LIN {X 0,Y 525.406,Z 288.21,A -85,B 0,C 180,E1 -4793.658,E2 -4793.658} C_VEL
LIN {X 0,Y 523.939,Z 280.222,A -85,B 0,C 180,E1 -4794.968,E2 -4794.968} C_VEL
LIN {X 0,Y 523.912,Z 280.228,A -85,B 0,C 180,E1 -4798.002,E2 -4798.002} C_VEL
LIN {X 0,Y 523.934,Z 280.223,A -85,B 0,C 180,E1 -4800.852,E2 -4800.852} C_VEL
LIN {X 0,Y 523.928,Z 280.222,A -85,B 0,C 180,E1 -4803.729,E2 -4803.729} C_VEL
LIN {X 0,Y 523.897,Z 280.231,A -85,B 0,C 180,E1 -4806.4,E2 -4806.4} C_VEL
LIN {X 0,Y 523.911,Z 280.22,A -85,B 0,C 180,E1 -4809.085,E2 -4809.085} C_VEL
LIN {X 0,Y 523.949,Z 280.218,A -85,B 0,C 180,E1 -4812.119,E2 -4812.119} C_VEL
LIN {X 0,Y 523.941,Z 280.216,A -85,B 0,C 180,E1 -4815.31,E2 -4815.31} C_VEL
LIN {X 0,Y 523.953,Z 280.22,A -85,B 0,C 180,E1 -4818.689,E2 -4818.689} C_VEL
LIN {X 0,Y 523.915,Z 280.22,A -85,B 0,C 180,E1 -4821.08,E2 -4821.08} C_VEL
LIN {X 0,Y 523.897,Z 280.221,A -85,B 0,C 180,E1 -4823.825,E2 -4823.825} C_VEL
LIN {X 0,Y 523.91,Z 280.227,A -85,B 0,C 180,E1 -4826.633,E2 -4826.633} C_VEL
LIN {X 0,Y 523.953,Z 280.214,A -85,B 0,C 180,E1 -4829.355,E2 -4829.355} C_VEL
LIN {X 0,Y 523.975,Z 280.213,A -85,B 0,C 180,E1 -4832.281,E2 -4832.281} C_VEL
LIN {X 0,Y 523.944,Z 280.223,A -85,B 0,C 180,E1 -4834.581,E2 -4834.581} C_VEL
LIN {X 0,Y 523.916,Z 280.218,A -85,B 0,C 180,E1 -4837.756,E2 -4837.756} C_VEL
LIN {X 0,Y 523.973,Z 280.213,A -85,B 0,C 180,E1 -4840.408,E2 -4840.408} C_VEL
LIN {X 0,Y 523.965,Z 280.219,A -85,B 0,C 180,E1 -4842.837,E2 -4842.837} C_VEL
LIN {X 0,Y 523.974,Z 280.214,A -85,B 0,C 180,E1 -4845.236,E2 -4845.236} C_VEL
LIN {X 0,Y 524.009,Z 280.208,A -85,B 0,C 180,E1 -4848.394,E2 -4848.394} C_VEL
LIN {X 0,Y 524.001,Z 280.207,A -85,B 0,C 180,E1 -4851.516,E2 -4851.516} C_VEL
LIN {X 0,Y 524.078,Z 280.204,A -85,B 0,C 180,E1 -4854.614,E2 -4854.614} C_VEL
LIN {X 0,Y 524.11,Z 280.194,A -85,B 0,C 180,E1 -4857.695,E2 -4857.695} C_VEL
LIN {X 0,Y 524.121,Z 280.199,A -85,B 0,C 180,E1 -4860.769,E2 -4860.769} C_VEL
LIN {X 0,Y 524.069,Z 280.206,A -85,B 0,C 180,E1 -4863.075,E2 -4863.075} C_VEL
LIN {X 0,Y 524.043,Z 280.202,A -85,B 0,C 180,E1 -4866.159,E2 -4866.159} C_VEL
LIN {X 0,Y 523.996,Z 280.213,A -85,B 0,C 180,E1 -4869.262,E2 -4869.262} C_VEL
LIN {X 0,Y 524,Z 280.208,A -85,B 0,C 180,E1 -4871.74,E2 -4871.74} C_VEL
LIN {X 0,Y 523.991,Z 280.217,A -85,B 0,C 180,E1 -4875.053,E2 -4875.053} C_VEL
LIN {X 0,Y 523.945,Z 280.214,A -85,B 0,C 180,E1 -4877.97,E2 -4877.97} C_VEL
LIN {X 0,Y 523.97,Z 280.212,A -85,B 0,C 180,E1 -4880.41,E2 -4880.41} C_VEL
LIN {X 0,Y 523.908,Z 280.224,A -85,B 0,C 180,E1 -4882.894,E2 -4882.894} C_VEL
LIN {X 0,Y 523.981,Z 280.21,A -85,B 0,C 180,E1 -4886.02,E2 -4886.02} C_VEL
LIN {X 0,Y 523.927,Z 280.221,A -85,B 0,C 180,E1 -4888.876,E2 -4888.876} C_VEL
LIN {X 0,Y 523.917,Z 280.221,A -85,B 0,C 180,E1 -4891.545,E2 -4891.545} C_VEL
LIN {X 0,Y 523.921,Z 280.217,A -85,B 0,C 180,E1 -4894.292,E2 -4894.292} C_VEL
LIN {X 0,Y 523.906,Z 280.226,A -85,B 0,C 180,E1 -4897.133,E2 -4897.133} C_VEL
LIN {X 0,Y 523.937,Z 280.216,A -85,B 0,C 180,E1 -4900.13,E2 -4900.13} C_VEL
LIN {X 0,Y 523.889,Z 280.229,A -85,B 0,C 180,E1 -4903.171,E2 -4903.171} C_VEL
LIN {X 0,Y 523.923,Z 280.222,A -85,B 0,C 180,E1 -4905.771,E2 -4905.771} C_VEL
LIN {X 0,Y 523.885,Z 280.225,A -85,B 0,C 180,E1 -4906.911,E2 -4906.911} C_VEL
LIN {X 0,Y 523.209,Z 280.314,A -85,B 0,C 180,E1 -4907.553,E2 -4907.553} C_VEL
LIN {X 0,Y 520.362,Z 280.666,A -85,B 0,C 180,E1 -4908.594,E2 -4908.594} C_VEL
LIN {X 0,Y 517.964,Z 280.968,A -85,B 0,C 180,E1 -4909.433,E2 -4909.433} C_VEL
LIN {X 0,Y 516.939,Z 281.09,A -85,B 0,C 180,E1 -4910.081,E2 -4910.081} C_VEL
LIN {X 0,Y 516.858,Z 281.099,A -85,B 0,C 180,E1 -4910.3,E2 -4910.3} C_VEL
LIN {X 0,Y 516.846,Z 281.107,A -85,B 0,C 180,E1 -4913.349,E2 -4913.349} C_VEL
LIN {X 0,Y 516.884,Z 281.097,A -85,B 0,C 180,E1 -4916.12,E2 -4916.12} C_VEL
LIN {X 0,Y 516.882,Z 281.099,A -85,B 0,C 180,E1 -4918.939,E2 -4918.939} C_VEL
LIN {X 0,Y 516.958,Z 281.096,A -85,B 0,C 180,E1 -4922.172,E2 -4922.172} C_VEL
LIN {X 0,Y 517.261,Z 286.094,A -85,B 0,C 180,E1 -4923.144,E2 -4923.144} C_VEL
LIN {X 0,Y 517.143,Z 299.715,A -85,B 0,C 180,E1 -4925.679,E2 -4925.679} C_VEL
LIN {X 0,Y 519.184,Z 310.941,A -85,B 0,C 180,E1 -4925.909,E2 -4925.909} C_VEL
LIN {X 0,Y 518.63,Z 406.558,A -85,B 0,C 180,E1 -4927.253,E2 -4927.253} C_VEL
LIN {X 0,Y 518.525,Z 420.061,A -85,B 0,C 180,E1 -4927.608,E2 -4927.608} C_VEL
LIN {X 0,Y 518.216,Z 432.786,A -85,B 0,C 180,E1 -4928.103,E2 -4928.103} C_VEL
LIN {X 0,Y 517.976,Z 444.369,A -85,B 0,C 180,E1 -4928.719,E2 -4928.719} C_VEL
LIN {X 0,Y 517.646,Z 456.07,A -85,B 0,C 180,E1 -4929.523,E2 -4929.523} C_VEL
LIN {X 0,Y 517.317,Z 466.867,A -85,B 0,C 180,E1 -4930.456,E2 -4930.456} C_VEL
LIN {X 0,Y 517.068,Z 475.452,A -85,B 0,C 180,E1 -4931.373,E2 -4931.373} C_VEL
LIN {X 0,Y 516.808,Z 484.688,A -85,B 0,C 180,E1 -4932.592,E2 -4932.592} C_VEL
LIN {X 0,Y 516.604,Z 492.063,A -85,B 0,C 180,E1 -4933.807,E2 -4933.807} C_VEL
LIN {X 0,Y 516.469,Z 498.021,A -85,B 0,C 180,E1 -4935.052,E2 -4935.052} C_VEL
LIN {X 0,Y 516.366,Z 502.404,A -85,B 0,C 180,E1 -4936.221,E2 -4936.221} C_VEL
LIN {X 0,Y 516.297,Z 505.806,A -85,B 0,C 180,E1 -4937.421,E2 -4937.421} C_VEL
LIN {X 0,Y 516.285,Z 508.091,A -85,B 0,C 180,E1 -4938.556,E2 -4938.556} C_VEL
LIN {X 0,Y 516.239,Z 509.597,A -85,B 0,C 180,E1 -4939.807,E2 -4939.807} C_VEL
LIN {X 0,Y 516.233,Z 510.026,A -85,B 0,C 180,E1 -4941.388,E2 -4941.388} C_VEL
LIN {X 0,Y 516.273,Z 509.658,A -85,B 0,C 180,E1 -4942.177,E2 -4942.177} C_VEL
LIN {X 0,Y 516.32,Z 508.057,A -85,B 0,C 180,E1 -4943.547,E2 -4943.547} C_VEL
LIN {X 0,Y 516.32,Z 506.098,A -85,B 0,C 180,E1 -4944.533,E2 -4944.533} C_VEL
LIN {X 0,Y 516.361,Z 502.896,A -85,B 0,C 180,E1 -4945.707,E2 -4945.707} C_VEL
LIN {X 0,Y 516.434,Z 498.648,A -85,B 0,C 180,E1 -4946.88,E2 -4946.88} C_VEL
LIN {X 0,Y 516.584,Z 492.239,A -85,B 0,C 180,E1 -4948.246,E2 -4948.246} C_VEL
LIN {X 0,Y 516.817,Z 485.213,A -85,B 0,C 180,E1 -4949.416,E2 -4949.416} C_VEL
LIN {X 0,Y 517.049,Z 476.502,A -85,B 0,C 180,E1 -4950.585,E2 -4950.585} C_VEL
LIN {X 0,Y 517.306,Z 466.62,A -85,B 0,C 180,E1 -4951.655,E2 -4951.655} C_VEL
LIN {X 0,Y 517.543,Z 456.543,A -85,B 0,C 180,E1 -4952.53,E2 -4952.53} C_VEL
LIN {X 0,Y 517.832,Z 445.389,A -85,B 0,C 180,E1 -4953.307,E2 -4953.307} C_VEL
LIN {X 0,Y 518.125,Z 434.797,A -85,B 0,C 180,E1 -4953.889,E2 -4953.889} C_VEL
LIN {X 0,Y 518.308,Z 423.339,A -85,B 0,C 180,E1 -4954.375,E2 -4954.375} C_VEL
LIN {X 0,Y 518.512,Z 411.153,A -85,B 0,C 180,E1 -4954.738,E2 -4954.738} C_VEL
LIN {X 0,Y 518.632,Z 395.767,A -85,B 0,C 180,E1 -4955.005,E2 -4955.005} C_VEL
LIN {X 0,Y 519.17,Z 310.059,A -85,B 0,C 180,E1 -4956.193,E2 -4956.193} C_VEL
LIN {X 0,Y 517.205,Z 299.754,A -85,B 0,C 180,E1 -4956.416,E2 -4956.416} C_VEL
LIN {X 0,Y 517.361,Z 285.225,A -85,B 0,C 180,E1 -4959.185,E2 -4959.185} C_VEL
LIN {X 0,Y 516.873,Z 281.104,A -85,B 0,C 180,E1 -4960.033,E2 -4960.033} C_VEL
LIN {X 0,Y 516.906,Z 281.1,A -85,B 0,C 180,E1 -4962.565,E2 -4962.565} C_VEL
LIN {X 0,Y 516.892,Z 281.093,A -85,B 0,C 180,E1 -4965.78,E2 -4965.78} C_VEL
LIN {X 0,Y 516.878,Z 281.097,A -85,B 0,C 180,E1 -4968.224,E2 -4968.224} C_VEL
LIN {X 0,Y 516.907,Z 281.1,A -85,B 0,C 180,E1 -4970.702,E2 -4970.702} C_VEL
LIN {X 0,Y 516.862,Z 281.1,A -85,B 0,C 180,E1 -4973.224,E2 -4973.224} C_VEL
LIN {X 0,Y 516.874,Z 281.096,A -85,B 0,C 180,E1 -4976.179,E2 -4976.179} C_VEL
LIN {X 0,Y 516.904,Z 281.096,A -85,B 0,C 180,E1 -4979.306,E2 -4979.306} C_VEL
LIN {X 0,Y 516.897,Z 281.095,A -85,B 0,C 180,E1 -4982.543,E2 -4982.543} C_VEL
LIN {X 0,Y 516.866,Z 281.102,A -85,B 0,C 180,E1 -4985.329,E2 -4985.329} C_VEL
LIN {X 0,Y 516.882,Z 281.094,A -85,B 0,C 180,E1 -4987.942,E2 -4987.942} C_VEL
LIN {X 0,Y 516.853,Z 281.1,A -85,B 0,C 180,E1 -4990.745,E2 -4990.745} C_VEL
LIN {X 0,Y 516.886,Z 281.095,A -85,B 0,C 180,E1 -4993.903,E2 -4993.903} C_VEL
LIN {X 0,Y 516.885,Z 281.094,A -85,B 0,C 180,E1 -4996.107,E2 -4996.107} C_VEL
LIN {X 0,Y 516.854,Z 281.105,A -85,B 0,C 180,E1 -4999.255,E2 -4999.255} C_VEL
LIN {X 0,Y 516.867,Z 281.097,A -85,B 0,C 180,E1 -5002.06,E2 -5002.06} C_VEL
LIN {X 0,Y 516.878,Z 281.099,A -85,B 0,C 180,E1 -5005.174,E2 -5005.174} C_VEL
LIN {X 0,Y 516.877,Z 281.098,A -85,B 0,C 180,E1 -5007.975,E2 -5007.975} C_VEL
LIN {X 0,Y 516.924,Z 281.089,A -85,B 0,C 180,E1 -5010.695,E2 -5010.695} C_VEL
LIN {X 0,Y 516.873,Z 281.103,A -85,B 0,C 180,E1 -5013.821,E2 -5013.821} C_VEL
LIN {X 0,Y 516.862,Z 281.096,A -85,B 0,C 180,E1 -5016.776,E2 -5016.776} C_VEL
LIN {X 0,Y 516.943,Z 281.094,A -85,B 0,C 180,E1 -5019.732,E2 -5019.732} C_VEL
LIN {X 0,Y 516.889,Z 281.094,A -85,B 0,C 180,E1 -5022.594,E2 -5022.594} C_VEL
LIN {X 0,Y 516.94,Z 281.087,A -85,B 0,C 180,E1 -5025.03,E2 -5025.03} C_VEL
LIN {X 0,Y 516.931,Z 281.094,A -85,B 0,C 180,E1 -5028.233,E2 -5028.233} C_VEL
LIN {X 0,Y 516.933,Z 281.089,A -85,B 0,C 180,E1 -5031.399,E2 -5031.399} C_VEL
LIN {X 0,Y 516.987,Z 281.085,A -85,B 0,C 180,E1 -5034.539,E2 -5034.539} C_VEL
LIN {X 0,Y 517.076,Z 281.072,A -85,B 0,C 180,E1 -5037.663,E2 -5037.663} C_VEL
LIN {X 0,Y 517.029,Z 281.079,A -85,B 0,C 180,E1 -5040.779,E2 -5040.779} C_VEL
LIN {X 0,Y 516.944,Z 281.087,A -85,B 0,C 180,E1 -5043.117,E2 -5043.117} C_VEL
LIN {X 0,Y 516.973,Z 281.089,A -85,B 0,C 180,E1 -5046.243,E2 -5046.243} C_VEL
LIN {X 0,Y 516.908,Z 281.091,A -85,B 0,C 180,E1 -5049.39,E2 -5049.39} C_VEL
LIN {X 0,Y 516.904,Z 281.101,A -85,B 0,C 180,E1 -5052.565,E2 -5052.565} C_VEL
LIN {X 0,Y 516.89,Z 281.093,A -85,B 0,C 180,E1 -5055.779,E2 -5055.779} C_VEL
LIN {X 0,Y 516.875,Z 281.098,A -85,B 0,C 180,E1 -5058.224,E2 -5058.224} C_VEL
LIN {X 0,Y 516.905,Z 281.101,A -85,B 0,C 180,E1 -5060.702,E2 -5060.702} C_VEL
LIN {X 0,Y 516.86,Z 281.1,A -85,B 0,C 180,E1 -5063.224,E2 -5063.224} C_VEL
LIN {X 0,Y 516.871,Z 281.096,A -85,B 0,C 180,E1 -5066.179,E2 -5066.179} C_VEL
LIN {X 0,Y 516.902,Z 281.095,A -85,B 0,C 180,E1 -5069.306,E2 -5069.306} C_VEL
LIN {X 0,Y 516.895,Z 281.095,A -85,B 0,C 180,E1 -5072.542,E2 -5072.542} C_VEL
LIN {X 0,Y 516.863,Z 281.102,A -85,B 0,C 180,E1 -5075.328,E2 -5075.328} C_VEL
LIN {X 0,Y 516.88,Z 281.095,A -85,B 0,C 180,E1 -5077.942,E2 -5077.942} C_VEL
LIN {X 0,Y 516.85,Z 281.101,A -85,B 0,C 180,E1 -5080.745,E2 -5080.745} C_VEL
LIN {X 0,Y 516.883,Z 281.095,A -85,B 0,C 180,E1 -5083.903,E2 -5083.903} C_VEL
LIN {X 0,Y 516.883,Z 281.094,A -85,B 0,C 180,E1 -5086.107,E2 -5086.107} C_VEL
LIN {X 0,Y 516.852,Z 281.106,A -85,B 0,C 180,E1 -5089.255,E2 -5089.255} C_VEL
LIN {X 0,Y 516.865,Z 281.097,A -85,B 0,C 180,E1 -5092.059,E2 -5092.059} C_VEL
LIN {X 0,Y 516.876,Z 281.099,A -85,B 0,C 180,E1 -5095.174,E2 -5095.174} C_VEL
LIN {X 0,Y 516.875,Z 281.099,A -85,B 0,C 180,E1 -5097.975,E2 -5097.975} C_VEL
LIN {X 0,Y 516.922,Z 281.091,A -85,B 0,C 180,E1 -5100.695,E2 -5100.695} C_VEL
LIN {X 0,Y 516.871,Z 281.105,A -85,B 0,C 180,E1 -5103.821,E2 -5103.821} C_VEL
LIN {X 0,Y 516.943,Z 281.212,A -85,B 0,C 180,E1 -5104.858,E2 -5104.858} C_VEL
LIN {X 0,Y 518.585,Z 290.856,A -85,B 0,C 180,E1 -5106.434,E2 -5106.434} C_VEL
LIN {X 0,Y 518.047,Z 310.917,A -85,B 0,C 180,E1 -5109.51,E2 -5109.51} C_VEL
LIN {X 0,Y 517.599,Z 329.015,A -85,B 0,C 180,E1 -5112.25,E2 -5112.25} C_VEL
LIN {X 0,Y 517.265,Z 344.925,A -85,B 0,C 180,E1 -5114.629,E2 -5114.629} C_VEL
LIN {X 0,Y 519.04,Z 358.237,A -85,B 0,C 180,E1 -5114.869,E2 -5114.869} C_VEL
LIN {X 0,Y 518.591,Z 453.375,A -85,B 0,C 180,E1 -5116.205,E2 -5116.205} C_VEL
LIN {X 0,Y 518.348,Z 466.709,A -85,B 0,C 180,E1 -5116.549,E2 -5116.549} C_VEL
LIN {X 0,Y 518.043,Z 480.041,A -85,B 0,C 180,E1 -5117.064,E2 -5117.064} C_VEL
LIN {X 0,Y 517.797,Z 491.638,A -85,B 0,C 180,E1 -5117.681,E2 -5117.681} C_VEL
LIN {X 0,Y 517.525,Z 502.87,A -85,B 0,C 180,E1 -5118.445,E2 -5118.445} C_VEL
LIN {X 0,Y 517.206,Z 513.346,A -85,B 0,C 180,E1 -5119.33,E2 -5119.33} C_VEL
LIN {X 0,Y 516.943,Z 521.914,A -85,B 0,C 180,E1 -5120.215,E2 -5120.215} C_VEL
LIN {X 0,Y 516.715,Z 529.823,A -85,B 0,C 180,E1 -5121.198,E2 -5121.198} C_VEL
LIN {X 0,Y 516.54,Z 537.55,A -85,B 0,C 180,E1 -5122.376,E2 -5122.376} C_VEL
LIN {X 0,Y 516.392,Z 544.673,A -85,B 0,C 180,E1 -5123.749,E2 -5123.749} C_VEL
LIN {X 0,Y 516.313,Z 549.413,A -85,B 0,C 180,E1 -5124.923,E2 -5124.923} C_VEL
LIN {X 0,Y 516.352,Z 553.039,A -85,B 0,C 180,E1 -5126.097,E2 -5126.097} C_VEL
LIN {X 0,Y 516.282,Z 554.905,A -85,B 0,C 180,E1 -5126.878,E2 -5126.878} C_VEL
LIN {X 0,Y 516.261,Z 556.306,A -85,B 0,C 180,E1 -5127.659,E2 -5127.659} C_VEL
LIN {X 0,Y 516.162,Z 557.911,A -85,B 0,C 180,E1 -5129.219,E2 -5129.219} C_VEL
LIN {X 0,Y 516.162,Z 558.128,A -85,B 0,C 180,E1 -5130,E2 -5130} C_VEL
LIN {X 0,Y 516.191,Z 557.301,A -85,B 0,C 180,E1 -5131.56,E2 -5131.56} C_VEL
LIN {X 0,Y 516.26,Z 556.304,A -85,B 0,C 180,E1 -5132.34,E2 -5132.34} C_VEL
LIN {X 0,Y 516.282,Z 554.903,A -85,B 0,C 180,E1 -5133.121,E2 -5133.121} C_VEL
LIN {X 0,Y 516.312,Z 551.955,A -85,B 0,C 180,E1 -5134.293,E2 -5134.293} C_VEL
LIN {X 0,Y 516.375,Z 547.966,A -85,B 0,C 180,E1 -5135.466,E2 -5135.466} C_VEL
LIN {X 0,Y 516.471,Z 542.086,A -85,B 0,C 180,E1 -5136.788,E2 -5136.788} C_VEL
LIN {X 0,Y 516.584,Z 535.126,A -85,B 0,C 180,E1 -5138.015,E2 -5138.015} C_VEL
LIN {X 0,Y 516.792,Z 526.812,A -85,B 0,C 180,E1 -5139.194,E2 -5139.194} C_VEL
LIN {X 0,Y 517.02,Z 518.293,A -85,B 0,C 180,E1 -5140.178,E2 -5140.178} C_VEL
LIN {X 0,Y 517.359,Z 507.773,A -85,B 0,C 180,E1 -5141.161,E2 -5141.161} C_VEL
LIN {X 0,Y 517.667,Z 496.279,A -85,B 0,C 180,E1 -5142.024,E2 -5142.024} C_VEL
LIN {X 0,Y 517.949,Z 485.966,A -85,B 0,C 180,E1 -5142.638,E2 -5142.638} C_VEL
LIN {X 0,Y 518.195,Z 474.267,A -85,B 0,C 180,E1 -5143.18,E2 -5143.18} C_VEL
LIN {X 0,Y 518.46,Z 461.713,A -85,B 0,C 180,E1 -5143.597,E2 -5143.597} C_VEL
LIN {X 0,Y 518.647,Z 448.998,A -85,B 0,C 180,E1 -5143.867,E2 -5143.867} C_VEL
LIN {X 0,Y 518.967,Z 356.025,A -85,B 0,C 180,E1 -5145.164,E2 -5145.164} C_VEL
LIN {X 0,Y 517.284,Z 344.745,A -85,B 0,C 180,E1 -5145.385,E2 -5145.385} C_VEL
LIN {X 0,Y 517.743,Z 323.23,A -85,B 0,C 180,E1 -5148.602,E2 -5148.602} C_VEL
LIN {X 0,Y 518.125,Z 305.573,A -85,B 0,C 180,E1 -5151.274,E2 -5151.274} C_VEL
LIN {X 0,Y 518.534,Z 290.622,A -85,B 0,C 180,E1 -5153.567,E2 -5153.567} C_VEL
LIN {X 0,Y 517.17,Z 282.406,A -85,B 0,C 180,E1 -5154.914,E2 -5154.914} C_VEL
LIN {X 0,Y 516.881,Z 281.101,A -85,B 0,C 180,E1 -5155.144,E2 -5155.144} C_VEL
LIN {X 0,Y 516.859,Z 281.109,A -85,B 0,C 180,E1 -5158.418,E2 -5158.418} C_VEL
LIN {X 0,Y 516.885,Z 281.099,A -85,B 0,C 180,E1 -5161.109,E2 -5161.109} C_VEL
LIN {X 0,Y 516.884,Z 281.102,A -85,B 0,C 180,E1 -5163.962,E2 -5163.962} C_VEL
LIN {X 0,Y 516.851,Z 281.103,A -85,B 0,C 180,E1 -5166.748,E2 -5166.748} C_VEL
LIN {X 0,Y 516.869,Z 281.097,A -85,B 0,C 180,E1 -5169.722,E2 -5169.722} C_VEL
LIN {X 0,Y 516.909,Z 281.092,A -85,B 0,C 180,E1 -5171.775,E2 -5171.775} C_VEL
LIN {X 0,Y 516.892,Z 281.096,A -85,B 0,C 180,E1 -5175.007,E2 -5175.007} C_VEL
LIN {X 0,Y 516.91,Z 281.1,A -85,B 0,C 180,E1 -5178.398,E2 -5178.398} C_VEL
LIN {X 0,Y 516.878,Z 281.095,A -85,B 0,C 180,E1 -5181.284,E2 -5181.284} C_VEL
LIN {X 0,Y 516.868,Z 281.101,A -85,B 0,C 180,E1 -5184.219,E2 -5184.219} C_VEL
LIN {X 0,Y 516.878,Z 281.097,A -85,B 0,C 180,E1 -5187.052,E2 -5187.052} C_VEL
LIN {X 0,Y 516.889,Z 281.093,A -85,B 0,C 180,E1 -5189.796,E2 -5189.796} C_VEL
LIN {X 0,Y 516.924,Z 281.094,A -85,B 0,C 180,E1 -5192.467,E2 -5192.467} C_VEL
LIN {X 0,Y 516.872,Z 281.097,A -85,B 0,C 180,E1 -5195.07,E2 -5195.07} C_VEL
LIN {X 0,Y 516.865,Z 281.097,A -85,B 0,C 180,E1 -5197.621,E2 -5197.621} C_VEL
LIN {X 0,Y 516.929,Z 281.088,A -85,B 0,C 180,E1 -5200.13,E2 -5200.13} C_VEL
LIN {X 0,Y 516.926,Z 281.096,A -85,B 0,C 180,E1 -5202.596,E2 -5202.596} C_VEL
LIN {X 0,Y 516.939,Z 281.093,A -85,B 0,C 180,E1 -5205.03,E2 -5205.03} C_VEL
LIN {X 0,Y 516.962,Z 281.084,A -85,B 0,C 180,E1 -5208.234,E2 -5208.234} C_VEL
LIN {X 0,Y 516.965,Z 281.084,A -85,B 0,C 180,E1 -5211.4,E2 -5211.4} C_VEL
LIN {X 0,Y 517.007,Z 281.079,A -85,B 0,C 180,E1 -5213.757,E2 -5213.757} C_VEL
LIN {X 0,Y 517.082,Z 281.07,A -85,B 0,C 180,E1 -5217.663,E2 -5217.663} C_VEL
LIN {X 0,Y 517.091,Z 281.074,A -85,B 0,C 180,E1 -5220.779,E2 -5220.779} C_VEL
LIN {X 0,Y 517.01,Z 281.085,A -85,B 0,C 180,E1 -5223.117,E2 -5223.117} C_VEL
LIN {X 0,Y 517.007,Z 281.079,A -85,B 0,C 180,E1 -5226.243,E2 -5226.243} C_VEL
LIN {X 0,Y 516.95,Z 281.089,A -85,B 0,C 180,E1 -5229.39,E2 -5229.39} C_VEL
LIN {X 0,Y 516.949,Z 281.086,A -85,B 0,C 180,E1 -5231.808,E2 -5231.808} C_VEL
LIN {X 0,Y 516.942,Z 281.096,A -85,B 0,C 180,E1 -5235.147,E2 -5235.147} C_VEL
LIN {X 0,Y 516.913,Z 281.09,A -85,B 0,C 180,E1 -5238.223,E2 -5238.223} C_VEL
LIN {X 0,Y 516.91,Z 281.094,A -85,B 0,C 180,E1 -5240.702,E2 -5240.702} C_VEL
LIN {X 0,Y 516.887,Z 281.094,A -85,B 0,C 180,E1 -5244.074,E2 -5244.074} C_VEL
LIN {X 0,Y 516.921,Z 281.091,A -85,B 0,C 180,E1 -5246.658,E2 -5246.658} C_VEL
LIN {X 0,Y 516.907,Z 281.096,A -85,B 0,C 180,E1 -5249.524,E2 -5249.524} C_VEL
LIN {X 0,Y 516.892,Z 281.092,A -85,B 0,C 180,E1 -5252.544,E2 -5252.544} C_VEL
LIN {X 0,Y 516.866,Z 281.103,A -85,B 0,C 180,E1 -5255.33,E2 -5255.33} C_VEL
LIN {X 0,Y 516.877,Z 281.095,A -85,B 0,C 180,E1 -5257.943,E2 -5257.943} C_VEL
LIN {X 0,Y 516.87,Z 281.097,A -85,B 0,C 180,E1 -5260.744,E2 -5260.744} C_VEL
LIN {X 0,Y 516.88,Z 281.098,A -85,B 0,C 180,E1 -5263.904,E2 -5263.904} C_VEL
LIN {X 0,Y 516.839,Z 281.103,A -85,B 0,C 180,E1 -5266.912,E2 -5266.912} C_VEL
LIN {X 0,Y 516.86,Z 281.106,A -85,B 0,C 180,E1 -5269.594,E2 -5269.594} C_VEL
LIN {X 0,Y 516.858,Z 281.099,A -85,B 0,C 180,E1 -5270.3,E2 -5270.3} C_VEL
LIN {X 0,Y 516.196,Z 281.185,A -85,B 0,C 180,E1 -5270.951,E2 -5270.951} C_VEL
LIN {X 0,Y 513.344,Z 281.544,A -85,B 0,C 180,E1 -5272.006,E2 -5272.006} C_VEL
LIN {X 0,Y 510.928,Z 281.848,A -85,B 0,C 180,E1 -5272.857,E2 -5272.857} C_VEL
LIN {X 0,Y 509.887,Z 281.975,A -85,B 0,C 180,E1 -5273.513,E2 -5273.513} C_VEL
LIN {X 0,Y 509.801,Z 281.982,A -85,B 0,C 180,E1 -5273.736,E2 -5273.736} C_VEL
LIN {X 0,Y 509.842,Z 281.973,A -85,B 0,C 180,E1 -5276.538,E2 -5276.538} C_VEL
LIN {X 0,Y 509.83,Z 281.982,A -85,B 0,C 180,E1 -5279.334,E2 -5279.334} C_VEL
LIN {X 0,Y 509.913,Z 282.133,A -85,B 0,C 180,E1 -5282.112,E2 -5282.112} C_VEL
LIN {X 0,Y 510.278,Z 286.613,A -85,B 0,C 180,E1 -5282.967,E2 -5282.967} C_VEL
LIN {X 0,Y 510.172,Z 299.959,A -85,B 0,C 180,E1 -5285.457,E2 -5285.457} C_VEL
LIN {X 0,Y 512.316,Z 311.121,A -85,B 0,C 180,E1 -5285.699,E2 -5285.699} C_VEL
LIN {X 0,Y 511.738,Z 407.246,A -85,B 0,C 180,E1 -5287.072,E2 -5287.072} C_VEL
LIN {X 0,Y 511.609,Z 420.675,A -85,B 0,C 180,E1 -5287.433,E2 -5287.433} C_VEL
LIN {X 0,Y 511.323,Z 433.669,A -85,B 0,C 180,E1 -5287.951,E2 -5287.951} C_VEL
LIN {X 0,Y 511.077,Z 444.279,A -85,B 0,C 180,E1 -5288.523,E2 -5288.523} C_VEL
LIN {X 0,Y 510.733,Z 455.065,A -85,B 0,C 180,E1 -5289.26,E2 -5289.26} C_VEL
LIN {X 0,Y 510.399,Z 465.824,A -85,B 0,C 180,E1 -5290.18,E2 -5290.18} C_VEL
LIN {X 0,Y 510.125,Z 474.67,A -85,B 0,C 180,E1 -5291.11,E2 -5291.11} C_VEL
LIN {X 0,Y 509.825,Z 482.664,A -85,B 0,C 180,E1 -5292.128,E2 -5292.128} C_VEL
LIN {X 0,Y 509.637,Z 490.54,A -85,B 0,C 180,E1 -5293.373,E2 -5293.373} C_VEL
LIN {X 0,Y 509.472,Z 495.821,A -85,B 0,C 180,E1 -5294.396,E2 -5294.396} C_VEL
LIN {X 0,Y 509.355,Z 500.889,A -85,B 0,C 180,E1 -5295.62,E2 -5295.62} C_VEL
LIN {X 0,Y 509.248,Z 504.771,A -85,B 0,C 180,E1 -5296.838,E2 -5296.838} C_VEL
LIN {X 0,Y 509.212,Z 508.391,A -85,B 0,C 180,E1 -5298.502,E2 -5298.502} C_VEL
LIN {X 0,Y 509.177,Z 509.812,A -85,B 0,C 180,E1 -5299.664,E2 -5299.664} C_VEL
LIN {X 0,Y 509.097,Z 510.313,A -85,B 0,C 180,E1 -5300.465,E2 -5300.465} C_VEL
LIN {X 0,Y 509.177,Z 510.064,A -85,B 0,C 180,E1 -5302.067,E2 -5302.067} C_VEL
LIN {X 0,Y 509.242,Z 508.431,A -85,B 0,C 180,E1 -5303.552,E2 -5303.552} C_VEL
LIN {X 0,Y 509.249,Z 506.703,A -85,B 0,C 180,E1 -5304.457,E2 -5304.457} C_VEL
LIN {X 0,Y 509.283,Z 503.61,A -85,B 0,C 180,E1 -5305.648,E2 -5305.648} C_VEL
LIN {X 0,Y 509.372,Z 499.475,A -85,B 0,C 180,E1 -5306.837,E2 -5306.837} C_VEL
LIN {X 0,Y 509.527,Z 493.194,A -85,B 0,C 180,E1 -5308.222,E2 -5308.222} C_VEL
LIN {X 0,Y 509.762,Z 486.363,A -85,B 0,C 180,E1 -5309.408,E2 -5309.408} C_VEL
LIN {X 0,Y 510.024,Z 477.831,A -85,B 0,C 180,E1 -5310.593,E2 -5310.593} C_VEL
LIN {X 0,Y 510.266,Z 469.123,A -85,B 0,C 180,E1 -5311.579,E2 -5311.579} C_VEL
LIN {X 0,Y 510.499,Z 459.592,A -85,B 0,C 180,E1 -5312.466,E2 -5312.466} C_VEL
LIN {X 0,Y 510.809,Z 449.165,A -85,B 0,C 180,E1 -5313.254,E2 -5313.254} C_VEL
LIN {X 0,Y 511.216,Z 437.538,A -85,B 0,C 180,E1 -5313.942,E2 -5313.942} C_VEL
LIN {X 0,Y 511.388,Z 425.574,A -85,B 0,C 180,E1 -5314.483,E2 -5314.483} C_VEL
LIN {X 0,Y 511.604,Z 412.481,A -85,B 0,C 180,E1 -5314.901,E2 -5314.901} C_VEL
LIN {X 0,Y 511.798,Z 399.525,A -85,B 0,C 180,E1 -5315.146,E2 -5315.146} C_VEL
LIN {X 0,Y 512.26,Z 310.506,A -85,B 0,C 180,E1 -5316.401,E2 -5316.401} C_VEL
LIN {X 0,Y 510.221,Z 299.977,A -85,B 0,C 180,E1 -5316.637,E2 -5316.637} C_VEL
LIN {X 0,Y 510.36,Z 285.969,A -85,B 0,C 180,E1 -5319.312,E2 -5319.312} C_VEL
LIN {X 0,Y 509.839,Z 281.98,A -85,B 0,C 180,E1 -5320.123,E2 -5320.123} C_VEL
LIN {X 0,Y 509.867,Z 281.976,A -85,B 0,C 180,E1 -5322.741,E2 -5322.741} C_VEL
LIN {X 0,Y 509.901,Z 281.965,A -85,B 0,C 180,E1 -5325.242,E2 -5325.242} C_VEL
LIN {X 0,Y 509.836,Z 281.978,A -85,B 0,C 180,E1 -5328.485,E2 -5328.485} C_VEL
LIN {X 0,Y 509.85,Z 281.976,A -85,B 0,C 180,E1 -5331.002,E2 -5331.002} C_VEL
LIN {X 0,Y 509.824,Z 281.974,A -85,B 0,C 180,E1 -5333.564,E2 -5333.564} C_VEL
LIN {X 0,Y 509.812,Z 281.977,A -85,B 0,C 180,E1 -5336.355,E2 -5336.355} C_VEL
LIN {X 0,Y 509.838,Z 281.979,A -85,B 0,C 180,E1 -5338.847,E2 -5338.847} C_VEL
LIN {X 0,Y 509.816,Z 281.976,A -85,B 0,C 180,E1 -5341.591,E2 -5341.591} C_VEL
LIN {X 0,Y 509.84,Z 281.972,A -85,B 0,C 180,E1 -5344.415,E2 -5344.415} C_VEL
LIN {X 0,Y 509.813,Z 281.981,A -85,B 0,C 180,E1 -5347.342,E2 -5347.342} C_VEL
LIN {X 0,Y 509.817,Z 281.974,A -85,B 0,C 180,E1 -5350.385,E2 -5350.385} C_VEL
LIN {X 0,Y 509.811,Z 281.98,A -85,B 0,C 180,E1 -5353.573,E2 -5353.573} C_VEL
LIN {X 0,Y 509.81,Z 281.975,A -85,B 0,C 180,E1 -5356.427,E2 -5356.427} C_VEL
LIN {X 0,Y 509.818,Z 281.98,A -85,B 0,C 180,E1 -5359.615,E2 -5359.615} C_VEL
LIN {X 0,Y 509.798,Z 281.977,A -85,B 0,C 180,E1 -5362.657,E2 -5362.657} C_VEL
LIN {X 0,Y 509.844,Z 281.976,A -85,B 0,C 180,E1 -5365.8,E2 -5365.8} C_VEL
LIN {X 0,Y 509.849,Z 281.97,A -85,B 0,C 180,E1 -5368.721,E2 -5368.721} C_VEL
LIN {X 0,Y 509.854,Z 281.972,A -85,B 0,C 180,E1 -5371.154,E2 -5371.154} C_VEL
LIN {X 0,Y 509.842,Z 281.979,A -85,B 0,C 180,E1 -5373.825,E2 -5373.825} C_VEL
LIN {X 0,Y 509.823,Z 281.975,A -85,B 0,C 180,E1 -5376.436,E2 -5376.436} C_VEL
LIN {X 0,Y 509.92,Z 281.971,A -85,B 0,C 180,E1 -5379.844,E2 -5379.844} C_VEL
LIN {X 0,Y 509.855,Z 281.97,A -85,B 0,C 180,E1 -5383.173,E2 -5383.173} C_VEL
LIN {X 0,Y 509.857,Z 281.973,A -85,B 0,C 180,E1 -5385.634,E2 -5385.634} C_VEL
LIN {X 0,Y 509.894,Z 281.973,A -85,B 0,C 180,E1 -5388.131,E2 -5388.131} C_VEL
LIN {X 0,Y 509.887,Z 281.966,A -85,B 0,C 180,E1 -5391.279,E2 -5391.279} C_VEL
LIN {X 0,Y 509.925,Z 281.963,A -85,B 0,C 180,E1 -5393.669,E2 -5393.669} C_VEL
LIN {X 0,Y 509.89,Z 281.966,A -85,B 0,C 180,E1 -5396.839,E2 -5396.839} C_VEL
LIN {X 0,Y 509.928,Z 281.967,A -85,B 0,C 180,E1 -5398.42,E2 -5398.42} C_VEL
LIN {X 0,Y 509.981,Z 281.956,A -85,B 0,C 180,E1 -5400.789,E2 -5400.789} C_VEL
LIN {X 0,Y 510.044,Z 281.955,A -85,B 0,C 180,E1 -5402.369,E2 -5402.369} C_VEL
LIN {X 0,Y 509.94,Z 281.959,A -85,B 0,C 180,E1 -5405.536,E2 -5405.536} C_VEL
LIN {X 0,Y 509.878,Z 281.969,A -85,B 0,C 180,E1 -5407.923,E2 -5407.923} C_VEL
LIN {X 0,Y 509.864,Z 281.97,A -85,B 0,C 180,E1 -5411.126,E2 -5411.126} C_VEL
LIN {X 0,Y 509.847,Z 281.97,A -85,B 0,C 180,E1 -5413.552,E2 -5413.552} C_VEL
LIN {X 0,Y 509.842,Z 281.972,A -85,B 0,C 180,E1 -5416.003,E2 -5416.003} C_VEL
LIN {X 0,Y 509.833,Z 281.978,A -85,B 0,C 180,E1 -5418.485,E2 -5418.485} C_VEL
LIN {X 0,Y 509.847,Z 281.976,A -85,B 0,C 180,E1 -5421.002,E2 -5421.002} C_VEL
LIN {X 0,Y 509.821,Z 281.974,A -85,B 0,C 180,E1 -5423.564,E2 -5423.564} C_VEL
LIN {X 0,Y 509.809,Z 281.977,A -85,B 0,C 180,E1 -5426.354,E2 -5426.354} C_VEL
LIN {X 0,Y 509.836,Z 281.98,A -85,B 0,C 180,E1 -5428.847,E2 -5428.847} C_VEL
LIN {X 0,Y 509.813,Z 281.976,A -85,B 0,C 180,E1 -5431.591,E2 -5431.591} C_VEL
LIN {X 0,Y 509.837,Z 281.973,A -85,B 0,C 180,E1 -5434.415,E2 -5434.415} C_VEL
LIN {X 0,Y 509.81,Z 281.981,A -85,B 0,C 180,E1 -5437.341,E2 -5437.341} C_VEL
LIN {X 0,Y 509.815,Z 281.975,A -85,B 0,C 180,E1 -5440.385,E2 -5440.385} C_VEL
LIN {X 0,Y 509.808,Z 281.98,A -85,B 0,C 180,E1 -5443.573,E2 -5443.573} C_VEL
LIN {X 0,Y 509.808,Z 281.975,A -85,B 0,C 180,E1 -5446.426,E2 -5446.426} C_VEL
LIN {X 0,Y 509.815,Z 281.98,A -85,B 0,C 180,E1 -5449.615,E2 -5449.615} C_VEL
LIN {X 0,Y 509.796,Z 281.977,A -85,B 0,C 180,E1 -5452.657,E2 -5452.657} C_VEL
LIN {X 0,Y 509.842,Z 281.976,A -85,B 0,C 180,E1 -5455.8,E2 -5455.8} C_VEL
LIN {X 0,Y 509.847,Z 281.971,A -85,B 0,C 180,E1 -5458.72,E2 -5458.72} C_VEL
LIN {X 0,Y 509.852,Z 281.974,A -85,B 0,C 180,E1 -5461.154,E2 -5461.154} C_VEL
LIN {X 0,Y 509.824,Z 281.98,A -85,B 0,C 180,E1 -5464.482,E2 -5464.482} C_VEL
LIN {X 0,Y 509.878,Z 282.159,A -85,B 0,C 180,E1 -5464.704,E2 -5464.704} C_VEL
LIN {X 0,Y 511.637,Z 291.838,A -85,B 0,C 180,E1 -5466.31,E2 -5466.31} C_VEL
LIN {X 0,Y 511.09,Z 311.411,A -85,B 0,C 180,E1 -5469.347,E2 -5469.347} C_VEL
LIN {X 0,Y 510.596,Z 330.097,A -85,B 0,C 180,E1 -5472.213,E2 -5472.213} C_VEL
LIN {X 0,Y 510.273,Z 344.814,A -85,B 0,C 180,E1 -5474.416,E2 -5474.416} C_VEL
LIN {X 0,Y 512.201,Z 359.249,A -85,B 0,C 180,E1 -5474.681,E2 -5474.681} C_VEL
LIN {X 0,Y 511.708,Z 453.028,A -85,B 0,C 180,E1 -5476.016,E2 -5476.016} C_VEL
LIN {X 0,Y 511.452,Z 465.604,A -85,B 0,C 180,E1 -5476.338,E2 -5476.338} C_VEL
LIN {X 0,Y 511.147,Z 478.577,A -85,B 0,C 180,E1 -5476.836,E2 -5476.836} C_VEL
LIN {X 0,Y 510.853,Z 490.007,A -85,B 0,C 180,E1 -5477.431,E2 -5477.431} C_VEL
LIN {X 0,Y 510.559,Z 501.237,A -85,B 0,C 180,E1 -5478.184,E2 -5478.184} C_VEL
LIN {X 0,Y 510.219,Z 511.937,A -85,B 0,C 180,E1 -5479.082,E2 -5479.082} C_VEL
LIN {X 0,Y 509.885,Z 521.581,A -85,B 0,C 180,E1 -5480.078,E2 -5480.078} C_VEL
LIN {X 0,Y 509.669,Z 529.491,A -85,B 0,C 180,E1 -5481.075,E2 -5481.075} C_VEL
LIN {X 0,Y 509.468,Z 537.219,A -85,B 0,C 180,E1 -5482.27,E2 -5482.27} C_VEL
LIN {X 0,Y 509.308,Z 544.343,A -85,B 0,C 180,E1 -5483.662,E2 -5483.662} C_VEL
LIN {X 0,Y 509.243,Z 549.084,A -85,B 0,C 180,E1 -5484.853,E2 -5484.853} C_VEL
LIN {X 0,Y 509.246,Z 552.709,A -85,B 0,C 180,E1 -5486.043,E2 -5486.043} C_VEL
LIN {X 0,Y 509.2,Z 554.576,A -85,B 0,C 180,E1 -5486.835,E2 -5486.835} C_VEL
LIN {X 0,Y 509.189,Z 555.978,A -85,B 0,C 180,E1 -5487.626,E2 -5487.626} C_VEL
LIN {X 0,Y 509.076,Z 557.582,A -85,B 0,C 180,E1 -5489.208,E2 -5489.208} C_VEL
LIN {X 0,Y 509.073,Z 557.798,A -85,B 0,C 180,E1 -5489.999,E2 -5489.999} C_VEL
LIN {X 0,Y 509.112,Z 556.971,A -85,B 0,C 180,E1 -5491.582,E2 -5491.582} C_VEL
LIN {X 0,Y 509.189,Z 555.974,A -85,B 0,C 180,E1 -5492.373,E2 -5492.373} C_VEL
LIN {X 0,Y 509.201,Z 554.571,A -85,B 0,C 180,E1 -5493.164,E2 -5493.164} C_VEL
LIN {X 0,Y 509.205,Z 551.621,A -85,B 0,C 180,E1 -5494.353,E2 -5494.353} C_VEL
LIN {X 0,Y 509.292,Z 547.631,A -85,B 0,C 180,E1 -5495.543,E2 -5495.543} C_VEL
LIN {X 0,Y 509.406,Z 541.596,A -85,B 0,C 180,E1 -5496.913,E2 -5496.913} C_VEL
LIN {X 0,Y 509.508,Z 534.788,A -85,B 0,C 180,E1 -5498.128,E2 -5498.128} C_VEL
LIN {X 0,Y 509.748,Z 526.473,A -85,B 0,C 180,E1 -5499.322,E2 -5499.322} C_VEL
LIN {X 0,Y 509.982,Z 517.952,A -85,B 0,C 180,E1 -5500.32,E2 -5500.32} C_VEL
LIN {X 0,Y 510.375,Z 507.431,A -85,B 0,C 180,E1 -5501.316,E2 -5501.316} C_VEL
LIN {X 0,Y 510.702,Z 495.935,A -85,B 0,C 180,E1 -5502.19,E2 -5502.19} C_VEL
LIN {X 0,Y 510.997,Z 485.619,A -85,B 0,C 180,E1 -5502.813,E2 -5502.813} C_VEL
LIN {X 0,Y 511.287,Z 473.918,A -85,B 0,C 180,E1 -5503.361,E2 -5503.361} C_VEL
LIN {X 0,Y 511.559,Z 461.358,A -85,B 0,C 180,E1 -5503.784,E2 -5503.784} C_VEL
LIN {X 0,Y 511.745,Z 448.632,A -85,B 0,C 180,E1 -5504.058,E2 -5504.058} C_VEL
LIN {X 0,Y 512.106,Z 356.866,A -85,B 0,C 180,E1 -5505.355,E2 -5505.355} C_VEL
LIN {X 0,Y 510.247,Z 344.438,A -85,B 0,C 180,E1 -5505.596,E2 -5505.596} C_VEL
LIN {X 0,Y 510.746,Z 322.885,A -85,B 0,C 180,E1 -5508.866,E2 -5508.866} C_VEL
LIN {X 0,Y 511.167,Z 306.614,A -85,B 0,C 180,E1 -5511.367,E2 -5511.367} C_VEL
LIN {X 0,Y 511.586,Z 291.697,A -85,B 0,C 180,E1 -5513.692,E2 -5513.692} C_VEL
LIN {X 0,Y 509.83,Z 281.979,A -85,B 0,C 180,E1 -5515.353,E2 -5515.353} C_VEL
LIN {X 0,Y 509.828,Z 281.984,A -85,B 0,C 180,E1 -5518.086,E2 -5518.086} C_VEL
LIN {X 0,Y 509.839,Z 281.981,A -85,B 0,C 180,E1 -5520.666,E2 -5520.666} C_VEL
LIN {X 0,Y 509.84,Z 281.977,A -85,B 0,C 180,E1 -5523.462,E2 -5523.462} C_VEL
LIN {X 0,Y 509.808,Z 281.986,A -85,B 0,C 180,E1 -5526.354,E2 -5526.354} C_VEL
LIN {X 0,Y 509.836,Z 281.972,A -85,B 0,C 180,E1 -5529.353,E2 -5529.353} C_VEL
LIN {X 0,Y 509.83,Z 281.982,A -85,B 0,C 180,E1 -5532.489,E2 -5532.489} C_VEL
LIN {X 0,Y 509.836,Z 281.973,A -85,B 0,C 180,E1 -5535.33,E2 -5535.33} C_VEL
LIN {X 0,Y 509.852,Z 281.977,A -85,B 0,C 180,E1 -5538.574,E2 -5538.574} C_VEL
LIN {X 0,Y 509.848,Z 281.971,A -85,B 0,C 180,E1 -5541.786,E2 -5541.786} C_VEL
LIN {X 0,Y 509.827,Z 281.98,A -85,B 0,C 180,E1 -5544.622,E2 -5544.622} C_VEL
LIN {X 0,Y 509.857,Z 281.969,A -85,B 0,C 180,E1 -5547.481,E2 -5547.481} C_VEL
LIN {X 0,Y 509.855,Z 281.973,A -85,B 0,C 180,E1 -5550.273,E2 -5550.273} C_VEL
LIN {X 0,Y 509.882,Z 281.971,A -85,B 0,C 180,E1 -5552.944,E2 -5552.944} C_VEL
LIN {X 0,Y 509.848,Z 281.968,A -85,B 0,C 180,E1 -5555.573,E2 -5555.573} C_VEL
LIN {X 0,Y 509.819,Z 281.976,A -85,B 0,C 180,E1 -5558.149,E2 -5558.149} C_VEL
LIN {X 0,Y 509.862,Z 281.975,A -85,B 0,C 180,E1 -5560.682,E2 -5560.682} C_VEL
LIN {X 0,Y 509.882,Z 281.968,A -85,B 0,C 180,E1 -5563.175,E2 -5563.175} C_VEL
LIN {X 0,Y 509.861,Z 281.97,A -85,B 0,C 180,E1 -5565.634,E2 -5565.634} C_VEL
LIN {X 0,Y 509.91,Z 281.972,A -85,B 0,C 180,E1 -5568.875,E2 -5568.875} C_VEL
LIN {X 0,Y 509.948,Z 281.957,A -85,B 0,C 180,E1 -5572.079,E2 -5572.079} C_VEL
LIN {X 0,Y 509.978,Z 281.958,A -85,B 0,C 180,E1 -5574.464,E2 -5574.464} C_VEL
LIN {X 0,Y 510.053,Z 281.946,A -85,B 0,C 180,E1 -5577.631,E2 -5577.631} C_VEL
LIN {X 0,Y 510.061,Z 281.95,A -85,B 0,C 180,E1 -5580.79,E2 -5580.79} C_VEL
LIN {X 0,Y 509.952,Z 281.963,A -85,B 0,C 180,E1 -5583.16,E2 -5583.16} C_VEL
LIN {X 0,Y 509.975,Z 281.955,A -85,B 0,C 180,E1 -5586.33,E2 -5586.33} C_VEL
LIN {X 0,Y 509.913,Z 281.967,A -85,B 0,C 180,E1 -5588.721,E2 -5588.721} C_VEL
LIN {X 0,Y 509.902,Z 281.964,A -85,B 0,C 180,E1 -5591.932,E2 -5591.932} C_VEL
LIN {X 0,Y 509.891,Z 281.972,A -85,B 0,C 180,E1 -5595.242,E2 -5595.242} C_VEL
LIN {X 0,Y 509.864,Z 281.968,A -85,B 0,C 180,E1 -5597.994,E2 -5597.994} C_VEL
LIN {X 0,Y 509.884,Z 281.967,A -85,B 0,C 180,E1 -5600.402,E2 -5600.402} C_VEL
LIN {X 0,Y 509.819,Z 281.978,A -85,B 0,C 180,E1 -5603.564,E2 -5603.564} C_VEL
LIN {X 0,Y 509.908,Z 281.963,A -85,B 0,C 180,E1 -5606.379,E2 -5606.379} C_VEL
LIN {X 0,Y 509.87,Z 281.971,A -85,B 0,C 180,E1 -5608.845,E2 -5608.845} C_VEL
LIN {X 0,Y 509.817,Z 281.977,A -85,B 0,C 180,E1 -5611.591,E2 -5611.591} C_VEL
LIN {X 0,Y 509.838,Z 281.972,A -85,B 0,C 180,E1 -5614.415,E2 -5614.415} C_VEL
LIN {X 0,Y 509.815,Z 281.982,A -85,B 0,C 180,E1 -5617.342,E2 -5617.342} C_VEL
LIN {X 0,Y 509.832,Z 281.973,A -85,B 0,C 180,E1 -5620.383,E2 -5620.383} C_VEL
LIN {X 0,Y 509.796,Z 281.983,A -85,B 0,C 180,E1 -5623.06,E2 -5623.06} C_VEL
LIN {X 0,Y 509.821,Z 281.979,A -85,B 0,C 180,E1 -5625.794,E2 -5625.794} C_VEL
LIN {X 0,Y 509.831,Z 281.974,A -85,B 0,C 180,E1 -5628.573,E2 -5628.573} C_VEL
LIN {X 0,Y 509.816,Z 281.98,A -85,B 0,C 180,E1 -5631.792,E2 -5631.792} C_VEL
LIN {X 0,Y 509.801,Z 281.982,A -85,B 0,C 180,E1 -5633.736,E2 -5633.736} C_VEL
LIN {X 0,Y 509.144,Z 282.06,A -85,B 0,C 180,E1 -5634.395,E2 -5634.395} C_VEL
LIN {X 0,Y 506.34,Z 282.415,A -85,B 0,C 180,E1 -5635.468,E2 -5635.468} C_VEL
LIN {X 0,Y 503.954,Z 282.711,A -85,B 0,C 180,E1 -5636.331,E2 -5636.331} C_VEL
LIN {X 0,Y 502.905,Z 282.84,A -85,B 0,C 180,E1 -5636.998,E2 -5636.998} C_VEL
LIN {X 0,Y 502.807,Z 282.851,A -85,B 0,C 180,E1 -5637.223,E2 -5637.223} C_VEL
LIN {X 0,Y 502.811,Z 282.855,A -85,B 0,C 180,E1 -5640.067,E2 -5640.067} C_VEL
LIN {X 0,Y 502.876,Z 282.957,A -85,B 0,C 180,E1 -5641.967,E2 -5641.967} C_VEL
LIN {X 0,Y 503.314,Z 287.189,A -85,B 0,C 180,E1 -5642.785,E2 -5642.785} C_VEL
LIN {X 0,Y 503.232,Z 300.367,A -85,B 0,C 180,E1 -5645.249,E2 -5645.249} C_VEL
LIN {X 0,Y 505.515,Z 312.691,A -85,B 0,C 180,E1 -5645.504,E2 -5645.504} C_VEL
LIN {X 0,Y 504.866,Z 407.27,A -85,B 0,C 180,E1 -5646.871,E2 -5646.871} C_VEL
LIN {X 0,Y 504.729,Z 420.98,A -85,B 0,C 180,E1 -5647.243,E2 -5647.243} C_VEL
LIN {X 0,Y 504.438,Z 433.415,A -85,B 0,C 180,E1 -5647.742,E2 -5647.742} C_VEL
LIN {X 0,Y 504.178,Z 444.174,A -85,B 0,C 180,E1 -5648.322,E2 -5648.322} C_VEL
LIN {X 0,Y 503.824,Z 454.525,A -85,B 0,C 180,E1 -5649.027,E2 -5649.027} C_VEL
LIN {X 0,Y 503.442,Z 465.87,A -85,B 0,C 180,E1 -5650.001,E2 -5650.001} C_VEL
LIN {X 0,Y 503.128,Z 475.675,A -85,B 0,C 180,E1 -5651.049,E2 -5651.049} C_VEL
LIN {X 0,Y 502.788,Z 483.602,A -85,B 0,C 180,E1 -5652.091,E2 -5652.091} C_VEL
LIN {X 0,Y 502.585,Z 491.294,A -85,B 0,C 180,E1 -5653.342,E2 -5653.342} C_VEL
LIN {X 0,Y 502.384,Z 497.416,A -85,B 0,C 180,E1 -5654.586,E2 -5654.586} C_VEL
LIN {X 0,Y 502.258,Z 502.212,A -85,B 0,C 180,E1 -5655.826,E2 -5655.826} C_VEL
LIN {X 0,Y 502.172,Z 505.841,A -85,B 0,C 180,E1 -5657.061,E2 -5657.061} C_VEL
LIN {X 0,Y 502.123,Z 508.705,A -85,B 0,C 180,E1 -5658.456,E2 -5658.456} C_VEL
LIN {X 0,Y 502.084,Z 510.017,A -85,B 0,C 180,E1 -5659.516,E2 -5659.516} C_VEL
LIN {X 0,Y 502.019,Z 510.591,A -85,B 0,C 180,E1 -5660.329,E2 -5660.329} C_VEL
LIN {X 0,Y 502.053,Z 510.736,A -85,B 0,C 180,E1 -5661.143,E2 -5661.143} C_VEL
LIN {X 0,Y 502.099,Z 510.468,A -85,B 0,C 180,E1 -5661.954,E2 -5661.954} C_VEL
LIN {X 0,Y 502.15,Z 508.782,A -85,B 0,C 180,E1 -5663.572,E2 -5663.572} C_VEL
LIN {X 0,Y 502.18,Z 507.309,A -85,B 0,C 180,E1 -5664.379,E2 -5664.379} C_VEL
LIN {X 0,Y 502.208,Z 504.323,A -85,B 0,C 180,E1 -5665.586,E2 -5665.586} C_VEL
LIN {X 0,Y 502.312,Z 500.301,A -85,B 0,C 180,E1 -5666.792,E2 -5666.792} C_VEL
LIN {X 0,Y 502.393,Z 495.145,A -85,B 0,C 180,E1 -5667.996,E2 -5667.996} C_VEL
LIN {X 0,Y 502.673,Z 488.667,A -85,B 0,C 180,E1 -5669.199,E2 -5669.199} C_VEL
LIN {X 0,Y 502.891,Z 480.66,A -85,B 0,C 180,E1 -5670.401,E2 -5670.401} C_VEL
LIN {X 0,Y 503.163,Z 472.493,A -85,B 0,C 180,E1 -5671.401,E2 -5671.401} C_VEL
LIN {X 0,Y 503.474,Z 462.511,A -85,B 0,C 180,E1 -5672.401,E2 -5672.401} C_VEL
LIN {X 0,Y 503.82,Z 451.244,A -85,B 0,C 180,E1 -5673.299,E2 -5673.299} C_VEL
LIN {X 0,Y 504.259,Z 440.159,A -85,B 0,C 180,E1 -5673.996,E2 -5673.996} C_VEL
LIN {X 0,Y 504.433,Z 427.828,A -85,B 0,C 180,E1 -5674.595,E2 -5674.595} C_VEL
LIN {X 0,Y 504.693,Z 414.61,A -85,B 0,C 180,E1 -5675.044,E2 -5675.044} C_VEL
LIN {X 0,Y 504.935,Z 401.548,A -85,B 0,C 180,E1 -5675.316,E2 -5675.316} C_VEL
LIN {X 0,Y 505.491,Z 311.693,A -85,B 0,C 180,E1 -5676.598,E2 -5676.598} C_VEL
LIN {X 0,Y 503.211,Z 300.232,A -85,B 0,C 180,E1 -5676.858,E2 -5676.858} C_VEL
LIN {X 0,Y 503.376,Z 287.809,A -85,B 0,C 180,E1 -5679.24,E2 -5679.24} C_VEL
LIN {X 0,Y 502.78,Z 282.86,A -85,B 0,C 180,E1 -5680.241,E2 -5680.241} C_VEL
LIN {X 0,Y 502.821,Z 282.851,A -85,B 0,C 180,E1 -5682.923,E2 -5682.923} C_VEL
LIN {X 0,Y 502.855,Z 282.842,A -85,B 0,C 180,E1 -5685.4,E2 -5685.4} C_VEL
LIN {X 0,Y 502.808,Z 282.857,A -85,B 0,C 180,E1 -5688.753,E2 -5688.753} C_VEL
LIN {X 0,Y 502.786,Z 282.852,A -85,B 0,C 180,E1 -5691.312,E2 -5691.312} C_VEL
LIN {X 0,Y 502.771,Z 282.852,A -85,B 0,C 180,E1 -5693.915,E2 -5693.915} C_VEL
LIN {X 0,Y 502.787,Z 282.854,A -85,B 0,C 180,E1 -5696.571,E2 -5696.571} C_VEL
LIN {X 0,Y 502.797,Z 282.849,A -85,B 0,C 180,E1 -5699.93,E2 -5699.93} C_VEL
LIN {X 0,Y 502.808,Z 282.857,A -85,B 0,C 180,E1 -5703.034,E2 -5703.034} C_VEL
LIN {X 0,Y 502.772,Z 282.852,A -85,B 0,C 180,E1 -5705.952,E2 -5705.952} C_VEL
LIN {X 0,Y 502.798,Z 282.855,A -85,B 0,C 180,E1 -5708.977,E2 -5708.977} C_VEL
LIN {X 0,Y 502.75,Z 282.855,A -85,B 0,C 180,E1 -5712.192,E2 -5712.192} C_VEL
LIN {X 0,Y 502.791,Z 282.857,A -85,B 0,C 180,E1 -5715.47,E2 -5715.47} C_VEL
LIN {X 0,Y 502.767,Z 282.855,A -85,B 0,C 180,E1 -5718.928,E2 -5718.928} C_VEL
LIN {X 0,Y 502.769,Z 282.854,A -85,B 0,C 180,E1 -5722.043,E2 -5722.043} C_VEL
LIN {X 0,Y 502.796,Z 282.851,A -85,B 0,C 180,E1 -5725.033,E2 -5725.033} C_VEL
LIN {X 0,Y 502.787,Z 282.854,A -85,B 0,C 180,E1 -5727.915,E2 -5727.915} C_VEL
LIN {X 0,Y 502.817,Z 282.846,A -85,B 0,C 180,E1 -5730.711,E2 -5730.711} C_VEL
LIN {X 0,Y 502.777,Z 282.857,A -85,B 0,C 180,E1 -5733.46,E2 -5733.46} C_VEL
LIN {X 0,Y 502.771,Z 282.857,A -85,B 0,C 180,E1 -5736.085,E2 -5736.085} C_VEL
LIN {X 0,Y 502.786,Z 282.85,A -85,B 0,C 180,E1 -5738.689,E2 -5738.689} C_VEL
LIN {X 0,Y 502.815,Z 282.848,A -85,B 0,C 180,E1 -5741.247,E2 -5741.247} C_VEL
LIN {X 0,Y 502.842,Z 282.844,A -85,B 0,C 180,E1 -5744.664,E2 -5744.664} C_VEL
LIN {X 0,Y 502.874,Z 282.849,A -85,B 0,C 180,E1 -5748.043,E2 -5748.043} C_VEL
LIN {X 0,Y 502.85,Z 282.842,A -85,B 0,C 180,E1 -5751.156,E2 -5751.156} C_VEL
LIN {X 0,Y 502.875,Z 282.841,A -85,B 0,C 180,E1 -5753.58,E2 -5753.58} C_VEL
LIN {X 0,Y 502.836,Z 282.845,A -85,B 0,C 180,E1 -5756.795,E2 -5756.795} C_VEL
LIN {X 0,Y 502.897,Z 282.843,A -85,B 0,C 180,E1 -5758.398,E2 -5758.398} C_VEL
LIN {X 0,Y 502.934,Z 282.834,A -85,B 0,C 180,E1 -5760.8,E2 -5760.8} C_VEL
LIN {X 0,Y 503.012,Z 282.831,A -85,B 0,C 180,E1 -5762.402,E2 -5762.402} C_VEL
LIN {X 0,Y 502.897,Z 282.837,A -85,B 0,C 180,E1 -5765.614,E2 -5765.614} C_VEL
LIN {X 0,Y 502.85,Z 282.845,A -85,B 0,C 180,E1 -5768.034,E2 -5768.034} C_VEL
LIN {X 0,Y 502.839,Z 282.844,A -85,B 0,C 180,E1 -5771.284,E2 -5771.284} C_VEL
LIN {X 0,Y 502.831,Z 282.854,A -85,B 0,C 180,E1 -5774.571,E2 -5774.571} C_VEL
LIN {X 0,Y 502.802,Z 282.852,A -85,B 0,C 180,E1 -5777.069,E2 -5777.069} C_VEL
LIN {X 0,Y 502.809,Z 282.847,A -85,B 0,C 180,E1 -5779.6,E2 -5779.6} C_VEL
LIN {X 0,Y 502.806,Z 282.856,A -85,B 0,C 180,E1 -5782.702,E2 -5782.702} C_VEL
LIN {X 0,Y 502.772,Z 282.852,A -85,B 0,C 180,E1 -5785.679,E2 -5785.679} C_VEL
LIN {X 0,Y 502.773,Z 282.854,A -85,B 0,C 180,E1 -5788.377,E2 -5788.377} C_VEL
LIN {X 0,Y 502.786,Z 282.857,A -85,B 0,C 180,E1 -5791.144,E2 -5791.144} C_VEL
LIN {X 0,Y 502.789,Z 282.85,A -85,B 0,C 180,E1 -5793.995,E2 -5793.995} C_VEL
LIN {X 0,Y 502.767,Z 282.861,A -85,B 0,C 180,E1 -5797.175,E2 -5797.175} C_VEL
LIN {X 0,Y 502.772,Z 282.852,A -85,B 0,C 180,E1 -5800.017,E2 -5800.017} C_VEL
LIN {X 0,Y 502.75,Z 282.864,A -85,B 0,C 180,E1 -5803.234,E2 -5803.234} C_VEL
LIN {X 0,Y 502.781,Z 282.854,A -85,B 0,C 180,E1 -5805.66,E2 -5805.66} C_VEL
LIN {X 0,Y 502.766,Z 282.857,A -85,B 0,C 180,E1 -5809.012,E2 -5809.012} C_VEL
LIN {X 0,Y 502.766,Z 282.854,A -85,B 0,C 180,E1 -5812.043,E2 -5812.043} C_VEL
LIN {X 0,Y 502.794,Z 282.852,A -85,B 0,C 180,E1 -5815.033,E2 -5815.033} C_VEL
LIN {X 0,Y 502.785,Z 282.855,A -85,B 0,C 180,E1 -5817.915,E2 -5817.915} C_VEL
LIN {X 0,Y 502.815,Z 282.848,A -85,B 0,C 180,E1 -5820.711,E2 -5820.711} C_VEL
LIN {X 0,Y 502.774,Z 282.859,A -85,B 0,C 180,E1 -5823.46,E2 -5823.46} C_VEL
LIN {X 0,Y 502.819,Z 282.912,A -85,B 0,C 180,E1 -5824.517,E2 -5824.517} C_VEL
LIN {X 0,Y 504.646,Z 292.789,A -85,B 0,C 180,E1 -5826.179,E2 -5826.179} C_VEL
LIN {X 0,Y 504.137,Z 311.182,A -85,B 0,C 180,E1 -5829.071,E2 -5829.071} C_VEL
LIN {X 0,Y 503.63,Z 329.09,A -85,B 0,C 180,E1 -5831.854,E2 -5831.854} C_VEL
LIN {X 0,Y 503.243,Z 344.344,A -85,B 0,C 180,E1 -5834.191,E2 -5834.191} C_VEL
LIN {X 0,Y 505.353,Z 358.918,A -85,B 0,C 180,E1 -5834.468,E2 -5834.468} C_VEL
LIN {X 0,Y 504.808,Z 452.68,A -85,B 0,C 180,E1 -5835.821,E2 -5835.821} C_VEL
LIN {X 0,Y 504.533,Z 466.027,A -85,B 0,C 180,E1 -5836.173,E2 -5836.173} C_VEL
LIN {X 0,Y 504.176,Z 479.366,A -85,B 0,C 180,E1 -5836.702,E2 -5836.702} C_VEL
LIN {X 0,Y 503.854,Z 491.654,A -85,B 0,C 180,E1 -5837.379,E2 -5837.379} C_VEL
LIN {X 0,Y 503.511,Z 503.5,A -85,B 0,C 180,E1 -5838.221,E2 -5838.221} C_VEL
LIN {X 0,Y 503.153,Z 513.731,A -85,B 0,C 180,E1 -5839.13,E2 -5839.13} C_VEL
LIN {X 0,Y 502.811,Z 522.936,A -85,B 0,C 180,E1 -5840.141,E2 -5840.141} C_VEL
LIN {X 0,Y 502.541,Z 531.91,A -85,B 0,C 180,E1 -5841.353,E2 -5841.353} C_VEL
LIN {X 0,Y 502.346,Z 539.135,A -85,B 0,C 180,E1 -5842.564,E2 -5842.564} C_VEL
LIN {X 0,Y 502.235,Z 544.013,A -85,B 0,C 180,E1 -5843.572,E2 -5843.572} C_VEL
LIN {X 0,Y 502.174,Z 548.755,A -85,B 0,C 180,E1 -5844.78,E2 -5844.78} C_VEL
LIN {X 0,Y 502.141,Z 552.379,A -85,B 0,C 180,E1 -5845.987,E2 -5845.987} C_VEL
LIN {X 0,Y 502.12,Z 554.247,A -85,B 0,C 180,E1 -5846.79,E2 -5846.79} C_VEL
LIN {X 0,Y 502.12,Z 555.649,A -85,B 0,C 180,E1 -5847.593,E2 -5847.593} C_VEL
LIN {X 0,Y 501.992,Z 557.252,A -85,B 0,C 180,E1 -5849.197,E2 -5849.197} C_VEL
LIN {X 0,Y 501.987,Z 557.468,A -85,B 0,C 180,E1 -5849.999,E2 -5849.999} C_VEL
LIN {X 0,Y 502.036,Z 556.641,A -85,B 0,C 180,E1 -5851.604,E2 -5851.604} C_VEL
LIN {X 0,Y 502.12,Z 555.643,A -85,B 0,C 180,E1 -5852.406,E2 -5852.406} C_VEL
LIN {X 0,Y 502.122,Z 554.239,A -85,B 0,C 180,E1 -5853.209,E2 -5853.209} C_VEL
LIN {X 0,Y 502.103,Z 551.286,A -85,B 0,C 180,E1 -5854.415,E2 -5854.415} C_VEL
LIN {X 0,Y 502.208,Z 547.296,A -85,B 0,C 180,E1 -5855.621,E2 -5855.621} C_VEL
LIN {X 0,Y 502.332,Z 541.26,A -85,B 0,C 180,E1 -5857.011,E2 -5857.011} C_VEL
LIN {X 0,Y 502.459,Z 534.45,A -85,B 0,C 180,E1 -5858.242,E2 -5858.242} C_VEL
LIN {X 0,Y 502.713,Z 526.133,A -85,B 0,C 180,E1 -5859.454,E2 -5859.454} C_VEL
LIN {X 0,Y 502.966,Z 517.61,A -85,B 0,C 180,E1 -5860.465,E2 -5860.465} C_VEL
LIN {X 0,Y 503.391,Z 507.089,A -85,B 0,C 180,E1 -5861.475,E2 -5861.475} C_VEL
LIN {X 0,Y 503.738,Z 495.59,A -85,B 0,C 180,E1 -5862.362,E2 -5862.362} C_VEL
LIN {X 0,Y 504.05,Z 485.272,A -85,B 0,C 180,E1 -5862.992,E2 -5862.992} C_VEL
LIN {X 0,Y 504.333,Z 473.565,A -85,B 0,C 180,E1 -5863.549,E2 -5863.549} C_VEL
LIN {X 0,Y 504.692,Z 460.087,A -85,B 0,C 180,E1 -5864.001,E2 -5864.001} C_VEL
LIN {X 0,Y 504.895,Z 446.735,A -85,B 0,C 180,E1 -5864.278,E2 -5864.278} C_VEL
LIN {X 0,Y 505.322,Z 358.011,A -85,B 0,C 180,E1 -5865.545,E2 -5865.545} C_VEL
LIN {X 0,Y 503.231,Z 344.076,A -85,B 0,C 180,E1 -5865.823,E2 -5865.823} C_VEL
LIN {X 0,Y 503.802,Z 322.571,A -85,B 0,C 180,E1 -5869.136,E2 -5869.136} C_VEL
LIN {X 0,Y 504.336,Z 304.981,A -85,B 0,C 180,E1 -5871.886,E2 -5871.886} C_VEL
LIN {X 0,Y 504.634,Z 292.797,A -85,B 0,C 180,E1 -5873.82,E2 -5873.82} C_VEL
LIN {X 0,Y 502.787,Z 282.857,A -85,B 0,C 180,E1 -5875.539,E2 -5875.539} C_VEL
LIN {X 0,Y 502.794,Z 282.861,A -85,B 0,C 180,E1 -5878.375,E2 -5878.375} C_VEL
LIN {X 0,Y 502.792,Z 282.856,A -85,B 0,C 180,E1 -5881.143,E2 -5881.143} C_VEL
LIN {X 0,Y 502.787,Z 282.859,A -85,B 0,C 180,E1 -5883.995,E2 -5883.995} C_VEL
LIN {X 0,Y 502.763,Z 282.855,A -85,B 0,C 180,E1 -5887.175,E2 -5887.175} C_VEL
LIN {X 0,Y 502.783,Z 282.854,A -85,B 0,C 180,E1 -5890.015,E2 -5890.015} C_VEL
LIN {X 0,Y 502.801,Z 282.854,A -85,B 0,C 180,E1 -5892.199,E2 -5892.199} C_VEL
LIN {X 0,Y 502.783,Z 282.852,A -85,B 0,C 180,E1 -5895.47,E2 -5895.47} C_VEL
LIN {X 0,Y 502.817,Z 282.849,A -85,B 0,C 180,E1 -5898.934,E2 -5898.934} C_VEL
LIN {X 0,Y 502.79,Z 282.852,A -85,B 0,C 180,E1 -5902.046,E2 -5902.046} C_VEL
LIN {X 0,Y 502.793,Z 282.851,A -85,B 0,C 180,E1 -5905.034,E2 -5905.034} C_VEL
LIN {X 0,Y 502.779,Z 282.852,A -85,B 0,C 180,E1 -5907.915,E2 -5907.915} C_VEL
LIN {X 0,Y 502.82,Z 282.852,A -85,B 0,C 180,E1 -5910.712,E2 -5910.712} C_VEL
LIN {X 0,Y 502.859,Z 282.841,A -85,B 0,C 180,E1 -5913.439,E2 -5913.439} C_VEL
LIN {X 0,Y 502.772,Z 282.851,A -85,B 0,C 180,E1 -5916.085,E2 -5916.085} C_VEL
LIN {X 0,Y 502.78,Z 282.858,A -85,B 0,C 180,E1 -5918.689,E2 -5918.689} C_VEL
LIN {X 0,Y 502.827,Z 282.848,A -85,B 0,C 180,E1 -5921.248,E2 -5921.248} C_VEL
LIN {X 0,Y 502.82,Z 282.844,A -85,B 0,C 180,E1 -5923.767,E2 -5923.767} C_VEL
LIN {X 0,Y 502.828,Z 282.848,A -85,B 0,C 180,E1 -5926.255,E2 -5926.255} C_VEL
LIN {X 0,Y 502.874,Z 282.845,A -85,B 0,C 180,E1 -5928.717,E2 -5928.717} C_VEL
LIN {X 0,Y 502.898,Z 282.834,A -85,B 0,C 180,E1 -5931.967,E2 -5931.967} C_VEL
LIN {X 0,Y 502.934,Z 282.835,A -85,B 0,C 180,E1 -5934.387,E2 -5934.387} C_VEL
LIN {X 0,Y 503.022,Z 282.822,A -85,B 0,C 180,E1 -5937.598,E2 -5937.598} C_VEL
LIN {X 0,Y 503.025,Z 282.819,A -85,B 0,C 180,E1 -5940,E2 -5940} C_VEL
LIN {X 0,Y 503.022,Z 282.823,A -85,B 0,C 180,E1 -5942.402,E2 -5942.402} C_VEL
LIN {X 0,Y 502.934,Z 282.832,A -85,B 0,C 180,E1 -5945.614,E2 -5945.614} C_VEL
LIN {X 0,Y 502.899,Z 282.836,A -85,B 0,C 180,E1 -5948.034,E2 -5948.034} C_VEL
LIN {X 0,Y 502.874,Z 282.845,A -85,B 0,C 180,E1 -5951.284,E2 -5951.284} C_VEL
LIN {X 0,Y 502.842,Z 282.845,A -85,B 0,C 180,E1 -5954.571,E2 -5954.571} C_VEL
LIN {X 0,Y 502.82,Z 282.845,A -85,B 0,C 180,E1 -5957.909,E2 -5957.909} C_VEL
LIN {X 0,Y 502.827,Z 282.847,A -85,B 0,C 180,E1 -5960.537,E2 -5960.537} C_VEL
LIN {X 0,Y 502.785,Z 282.857,A -85,B 0,C 180,E1 -5963.041,E2 -5963.041} C_VEL
LIN {X 0,Y 502.818,Z 282.849,A -85,B 0,C 180,E1 -5965.677,E2 -5965.677} C_VEL
LIN {X 0,Y 502.835,Z 282.844,A -85,B 0,C 180,E1 -5968.373,E2 -5968.373} C_VEL
LIN {X 0,Y 502.79,Z 282.853,A -85,B 0,C 180,E1 -5971.499,E2 -5971.499} C_VEL
LIN {X 0,Y 502.789,Z 282.851,A -85,B 0,C 180,E1 -5973.996,E2 -5973.996} C_VEL
LIN {X 0,Y 502.776,Z 282.859,A -85,B 0,C 180,E1 -5977.178,E2 -5977.178} C_VEL
LIN {X 0,Y 502.781,Z 282.852,A -85,B 0,C 180,E1 -5980.016,E2 -5980.016} C_VEL
LIN {X 0,Y 502.77,Z 282.853,A -85,B 0,C 180,E1 -5982.196,E2 -5982.196} C_VEL
LIN {X 0,Y 502.785,Z 282.858,A -85,B 0,C 180,E1 -5985.471,E2 -5985.471} C_VEL
LIN {X 0,Y 502.78,Z 282.856,A -85,B 0,C 180,E1 -5987.86,E2 -5987.86} C_VEL
LIN {X 0,Y 502.783,Z 282.856,A -85,B 0,C 180,E1 -5991.023,E2 -5991.023} C_VEL
LIN {X 0,Y 502.769,Z 282.853,A -85,B 0,C 180,E1 -5994.171,E2 -5994.171} C_VEL
LIN {X 0,Y 502.807,Z 282.851,A -85,B 0,C 180,E1 -5997.223,E2 -5997.223} C_VEL
LIN {X 0,Y 502.103,Z 282.943,A -85,B 0,C 180,E1 -5997.892,E2 -5997.892} C_VEL
LIN {X 0,Y 499.237,Z 283.298,A -85,B 0,C 180,E1 -5998.978,E2 -5998.978} C_VEL
LIN {X 0,Y 496.842,Z 283.599,A -85,B 0,C 180,E1 -5999.852,E2 -5999.852} C_VEL
LIN {X 0,Y 495.826,Z 283.723,A -85,B 0,C 180,E1 -6000.528,E2 -6000.528} C_VEL
LIN {X 0,Y 495.748,Z 283.733,A -85,B 0,C 180,E1 -6000.757,E2 -6000.757} C_VEL
LIN {X 0,Y 495.855,Z 283.904,A -85,B 0,C 180,E1 -6001.828,E2 -6001.828} C_VEL
LIN {X 0,Y 496.34,Z 289.035,A -85,B 0,C 180,E1 -6002.83,E2 -6002.83} C_VEL
LIN {X 0,Y 496.253,Z 300.574,A -85,B 0,C 180,E1 -6005.01,E2 -6005.01} C_VEL
LIN {X 0,Y 498.629,Z 312.482,A -85,B 0,C 180,E1 -6005.27,E2 -6005.27} C_VEL
LIN {X 0,Y 498.012,Z 407.801,A -85,B 0,C 180,E1 -6006.673,E2 -6006.673} C_VEL
LIN {X 0,Y 497.861,Z 421.392,A -85,B 0,C 180,E1 -6007.048,E2 -6007.048} C_VEL
LIN {X 0,Y 497.532,Z 434.353,A -85,B 0,C 180,E1 -6007.58,E2 -6007.58} C_VEL
LIN {X 0,Y 497.228,Z 445.765,A -85,B 0,C 180,E1 -6008.222,E2 -6008.222} C_VEL
LIN {X 0,Y 496.838,Z 456.718,A -85,B 0,C 180,E1 -6009.005,E2 -6009.005} C_VEL
LIN {X 0,Y 496.454,Z 467.03,A -85,B 0,C 180,E1 -6009.923,E2 -6009.923} C_VEL
LIN {X 0,Y 496.099,Z 476.641,A -85,B 0,C 180,E1 -6010.985,E2 -6010.985} C_VEL
LIN {X 0,Y 495.761,Z 484.45,A -85,B 0,C 180,E1 -6012.042,E2 -6012.042} C_VEL
LIN {X 0,Y 495.541,Z 492.049,A -85,B 0,C 180,E1 -6013.31,E2 -6013.31} C_VEL
LIN {X 0,Y 495.343,Z 497.168,A -85,B 0,C 180,E1 -6014.362,E2 -6014.362} C_VEL
LIN {X 0,Y 495.203,Z 502.089,A -85,B 0,C 180,E1 -6015.62,E2 -6015.62} C_VEL
LIN {X 0,Y 495.094,Z 505.834,A -85,B 0,C 180,E1 -6016.873,E2 -6016.873} C_VEL
LIN {X 0,Y 495.046,Z 509.008,A -85,B 0,C 180,E1 -6018.401,E2 -6018.401} C_VEL
LIN {X 0,Y 494.995,Z 510.222,A -85,B 0,C 180,E1 -6019.364,E2 -6019.364} C_VEL
LIN {X 0,Y 494.961,Z 511.078,A -85,B 0,C 180,E1 -6021.015,E2 -6021.015} C_VEL
LIN {X 0,Y 495,Z 510.874,A -85,B 0,C 180,E1 -6021.838,E2 -6021.838} C_VEL
LIN {X 0,Y 495.079,Z 509.286,A -85,B 0,C 180,E1 -6023.48,E2 -6023.48} C_VEL
LIN {X 0,Y 495.114,Z 507.906,A -85,B 0,C 180,E1 -6024.298,E2 -6024.298} C_VEL
LIN {X 0,Y 495.116,Z 505.016,A -85,B 0,C 180,E1 -6025.523,E2 -6025.523} C_VEL
LIN {X 0,Y 495.254,Z 501.1,A -85,B 0,C 180,E1 -6026.747,E2 -6026.747} C_VEL
LIN {X 0,Y 495.327,Z 496.082,A -85,B 0,C 180,E1 -6027.968,E2 -6027.968} C_VEL
LIN {X 0,Y 495.622,Z 489.754,A -85,B 0,C 180,E1 -6029.188,E2 -6029.188} C_VEL
LIN {X 0,Y 495.848,Z 481.904,A -85,B 0,C 180,E1 -6030.407,E2 -6030.407} C_VEL
LIN {X 0,Y 496.231,Z 472.153,A -85,B 0,C 180,E1 -6031.624,E2 -6031.624} C_VEL
LIN {X 0,Y 496.527,Z 461.969,A -85,B 0,C 180,E1 -6032.637,E2 -6032.637} C_VEL
LIN {X 0,Y 496.922,Z 450.504,A -85,B 0,C 180,E1 -6033.548,E2 -6033.548} C_VEL
LIN {X 0,Y 497.397,Z 439.125,A -85,B 0,C 180,E1 -6034.255,E2 -6034.255} C_VEL
LIN {X 0,Y 497.584,Z 427.458,A -85,B 0,C 180,E1 -6034.811,E2 -6034.811} C_VEL
LIN {X 0,Y 497.81,Z 414.868,A -85,B 0,C 180,E1 -6035.24,E2 -6035.24} C_VEL
LIN {X 0,Y 498.063,Z 401.746,A -85,B 0,C 180,E1 -6035.517,E2 -6035.517} C_VEL
LIN {X 0,Y 498.597,Z 312.262,A -85,B 0,C 180,E1 -6036.811,E2 -6036.811} C_VEL
LIN {X 0,Y 496.226,Z 300.481,A -85,B 0,C 180,E1 -6037.083,E2 -6037.083} C_VEL
LIN {X 0,Y 496.381,Z 288.593,A -85,B 0,C 180,E1 -6039.371,E2 -6039.371} C_VEL
LIN {X 0,Y 495.739,Z 283.737,A -85,B 0,C 180,E1 -6040.363,E2 -6040.363} C_VEL
LIN {X 0,Y 495.791,Z 283.729,A -85,B 0,C 180,E1 -6042.277,E2 -6042.277} C_VEL
LIN {X 0,Y 495.811,Z 283.719,A -85,B 0,C 180,E1 -6045.624,E2 -6045.624} C_VEL
LIN {X 0,Y 495.769,Z 283.729,A -85,B 0,C 180,E1 -6049.03,E2 -6049.03} C_VEL
LIN {X 0,Y 495.746,Z 283.727,A -85,B 0,C 180,E1 -6051.629,E2 -6051.629} C_VEL
LIN {X 0,Y 495.717,Z 283.732,A -85,B 0,C 180,E1 -6054.277,E2 -6054.277} C_VEL
LIN {X 0,Y 495.734,Z 283.737,A -85,B 0,C 180,E1 -6056.979,E2 -6056.979} C_VEL
LIN {X 0,Y 495.748,Z 283.727,A -85,B 0,C 180,E1 -6060.143,E2 -6060.143} C_VEL
LIN {X 0,Y 495.757,Z 283.732,A -85,B 0,C 180,E1 -6063.237,E2 -6063.237} C_VEL
LIN {X 0,Y 495.717,Z 283.731,A -85,B 0,C 180,E1 -6066.087,E2 -6066.087} C_VEL
LIN {X 0,Y 495.762,Z 283.728,A -85,B 0,C 180,E1 -6068.767,E2 -6068.767} C_VEL
LIN {X 0,Y 495.728,Z 283.731,A -85,B 0,C 180,E1 -6071.785,E2 -6071.785} C_VEL
LIN {X 0,Y 495.742,Z 283.734,A -85,B 0,C 180,E1 -6075.141,E2 -6075.141} C_VEL
LIN {X 0,Y 495.728,Z 283.729,A -85,B 0,C 180,E1 -6078.215,E2 -6078.215} C_VEL
LIN {X 0,Y 495.744,Z 283.733,A -85,B 0,C 180,E1 -6081.235,E2 -6081.235} C_VEL
LIN {X 0,Y 495.747,Z 283.727,A -85,B 0,C 180,E1 -6084.462,E2 -6084.462} C_VEL
LIN {X 0,Y 495.757,Z 283.732,A -85,B 0,C 180,E1 -6087.404,E2 -6087.404} C_VEL
LIN {X 0,Y 495.767,Z 283.726,A -85,B 0,C 180,E1 -6090.253,E2 -6090.253} C_VEL
LIN {X 0,Y 495.743,Z 283.731,A -85,B 0,C 180,E1 -6093.271,E2 -6093.271} C_VEL
LIN {X 0,Y 495.744,Z 283.728,A -85,B 0,C 180,E1 -6096.612,E2 -6096.612} C_VEL
LIN {X 0,Y 495.784,Z 283.725,A -85,B 0,C 180,E1 -6099.324,E2 -6099.324} C_VEL
LIN {X 0,Y 495.784,Z 283.731,A -85,B 0,C 180,E1 -6101.828,E2 -6101.828} C_VEL
LIN {X 0,Y 495.785,Z 283.723,A -85,B 0,C 180,E1 -6105.217,E2 -6105.217} C_VEL
LIN {X 0,Y 495.826,Z 283.719,A -85,B 0,C 180,E1 -6108.554,E2 -6108.554} C_VEL
LIN {X 0,Y 495.817,Z 283.724,A -85,B 0,C 180,E1 -6111.851,E2 -6111.851} C_VEL
LIN {X 0,Y 495.857,Z 283.72,A -85,B 0,C 180,E1 -6114.306,E2 -6114.306} C_VEL
LIN {X 0,Y 495.979,Z 283.699,A -85,B 0,C 180,E1 -6117.563,E2 -6117.563} C_VEL
LIN {X 0,Y 495.975,Z 283.703,A -85,B 0,C 180,E1 -6120,E2 -6120} C_VEL
LIN {X 0,Y 495.978,Z 283.706,A -85,B 0,C 180,E1 -6122.436,E2 -6122.436} C_VEL
LIN {X 0,Y 495.856,Z 283.714,A -85,B 0,C 180,E1 -6125.694,E2 -6125.694} C_VEL
LIN {X 0,Y 495.814,Z 283.723,A -85,B 0,C 180,E1 -6128.149,E2 -6128.149} C_VEL
LIN {X 0,Y 495.824,Z 283.717,A -85,B 0,C 180,E1 -6131.446,E2 -6131.446} C_VEL
LIN {X 0,Y 495.782,Z 283.729,A -85,B 0,C 180,E1 -6134.783,E2 -6134.783} C_VEL
LIN {X 0,Y 495.742,Z 283.729,A -85,B 0,C 180,E1 -6137.32,E2 -6137.32} C_VEL
LIN {X 0,Y 495.76,Z 283.726,A -85,B 0,C 180,E1 -6139.891,E2 -6139.891} C_VEL
LIN {X 0,Y 495.762,Z 283.734,A -85,B 0,C 180,E1 -6142.86,E2 -6142.86} C_VEL
LIN {X 0,Y 495.714,Z 283.731,A -85,B 0,C 180,E1 -6146.072,E2 -6146.072} C_VEL
LIN {X 0,Y 495.723,Z 283.738,A -85,B 0,C 180,E1 -6148.818,E2 -6148.818} C_VEL
LIN {X 0,Y 495.751,Z 283.727,A -85,B 0,C 180,E1 -6151.723,E2 -6151.723} C_VEL
LIN {X 0,Y 495.762,Z 283.729,A -85,B 0,C 180,E1 -6154.692,E2 -6154.692} C_VEL
LIN {X 0,Y 495.723,Z 283.733,A -85,B 0,C 180,E1 -6157.562,E2 -6157.562} C_VEL
LIN {X 0,Y 495.745,Z 283.727,A -85,B 0,C 180,E1 -6160.044,E2 -6160.044} C_VEL
LIN {X 0,Y 495.698,Z 283.737,A -85,B 0,C 180,E1 -6162.886,E2 -6162.886} C_VEL
LIN {X 0,Y 495.725,Z 283.731,A -85,B 0,C 180,E1 -6165.997,E2 -6165.997} C_VEL
LIN {X 0,Y 495.729,Z 283.738,A -85,B 0,C 180,E1 -6169.296,E2 -6169.296} C_VEL
LIN {X 0,Y 495.726,Z 283.739,A -85,B 0,C 180,E1 -6171.406,E2 -6171.406} C_VEL
LIN {X 0,Y 495.744,Z 283.727,A -85,B 0,C 180,E1 -6174.461,E2 -6174.461} C_VEL
LIN {X 0,Y 495.755,Z 283.733,A -85,B 0,C 180,E1 -6177.404,E2 -6177.404} C_VEL
LIN {X 0,Y 495.765,Z 283.728,A -85,B 0,C 180,E1 -6180.253,E2 -6180.253} C_VEL
LIN {X 0,Y 495.741,Z 283.734,A -85,B 0,C 180,E1 -6183.27,E2 -6183.27} C_VEL
LIN {X 0,Y 495.797,Z 283.817,A -85,B 0,C 180,E1 -6184.355,E2 -6184.355} C_VEL
LIN {X 0,Y 497.661,Z 293.717,A -85,B 0,C 180,E1 -6186.045,E2 -6186.045} C_VEL
LIN {X 0,Y 497.204,Z 310.582,A -85,B 0,C 180,E1 -6188.734,E2 -6188.734} C_VEL
LIN {X 0,Y 496.665,Z 328.589,A -85,B 0,C 180,E1 -6191.571,E2 -6191.571} C_VEL
LIN {X 0,Y 496.232,Z 343.914,A -85,B 0,C 180,E1 -6193.963,E2 -6193.963} C_VEL
LIN {X 0,Y 498.504,Z 360.088,A -85,B 0,C 180,E1 -6194.273,E2 -6194.273} C_VEL
LIN {X 0,Y 497.924,Z 452.298,A -85,B 0,C 180,E1 -6195.621,E2 -6195.621} C_VEL
LIN {X 0,Y 497.611,Z 465.669,A -85,B 0,C 180,E1 -6195.977,E2 -6195.977} C_VEL
LIN {X 0,Y 497.257,Z 479.023,A -85,B 0,C 180,E1 -6196.514,E2 -6196.514} C_VEL
LIN {X 0,Y 496.928,Z 490.202,A -85,B 0,C 180,E1 -6197.127,E2 -6197.127} C_VEL
LIN {X 0,Y 496.569,Z 501.867,A -85,B 0,C 180,E1 -6197.95,E2 -6197.95} C_VEL
LIN {X 0,Y 496.139,Z 512.345,A -85,B 0,C 180,E1 -6198.871,E2 -6198.871} C_VEL
LIN {X 0,Y 495.827,Z 520.916,A -85,B 0,C 180,E1 -6199.794,E2 -6199.794} C_VEL
LIN {X 0,Y 495.555,Z 528.827,A -85,B 0,C 180,E1 -6200.819,E2 -6200.819} C_VEL
LIN {X 0,Y 495.331,Z 536.557,A -85,B 0,C 180,E1 -6202.048,E2 -6202.048} C_VEL
LIN {X 0,Y 495.164,Z 543.683,A -85,B 0,C 180,E1 -6203.48,E2 -6203.48} C_VEL
LIN {X 0,Y 495.106,Z 548.426,A -85,B 0,C 180,E1 -6204.705,E2 -6204.705} C_VEL
LIN {X 0,Y 495.035,Z 552.048,A -85,B 0,C 180,E1 -6205.929,E2 -6205.929} C_VEL
LIN {X 0,Y 495.042,Z 553.919,A -85,B 0,C 180,E1 -6206.744,E2 -6206.744} C_VEL
LIN {X 0,Y 495.024,Z 555.32,A -85,B 0,C 180,E1 -6207.558,E2 -6207.558} C_VEL
LIN {X 0,Y 494.912,Z 556.923,A -85,B 0,C 180,E1 -6209.186,E2 -6209.186} C_VEL
LIN {X 0,Y 494.905,Z 557.139,A -85,B 0,C 180,E1 -6209.999,E2 -6209.999} C_VEL
LIN {X 0,Y 494.963,Z 556.31,A -85,B 0,C 180,E1 -6211.627,E2 -6211.627} C_VEL
LIN {X 0,Y 495.024,Z 555.311,A -85,B 0,C 180,E1 -6212.441,E2 -6212.441} C_VEL
LIN {X 0,Y 495.045,Z 553.907,A -85,B 0,C 180,E1 -6213.255,E2 -6213.255} C_VEL
LIN {X 0,Y 495.008,Z 550.953,A -85,B 0,C 180,E1 -6214.478,E2 -6214.478} C_VEL
LIN {X 0,Y 495.124,Z 546.961,A -85,B 0,C 180,E1 -6215.702,E2 -6215.702} C_VEL
LIN {X 0,Y 495.255,Z 540.821,A -85,B 0,C 180,E1 -6217.132,E2 -6217.132} C_VEL
LIN {X 0,Y 495.414,Z 534.112,A -85,B 0,C 180,E1 -6218.36,E2 -6218.36} C_VEL
LIN {X 0,Y 495.673,Z 525.793,A -85,B 0,C 180,E1 -6219.59,E2 -6219.59} C_VEL
LIN {X 0,Y 495.965,Z 517.269,A -85,B 0,C 180,E1 -6220.615,E2 -6220.615} C_VEL
LIN {X 0,Y 496.401,Z 506.745,A -85,B 0,C 180,E1 -6221.639,E2 -6221.639} C_VEL
LIN {X 0,Y 496.763,Z 495.374,A -85,B 0,C 180,E1 -6222.529,E2 -6222.529} C_VEL
LIN {X 0,Y 497.168,Z 483.005,A -85,B 0,C 180,E1 -6223.28,E2 -6223.28} C_VEL
LIN {X 0,Y 497.487,Z 470.632,A -85,B 0,C 180,E1 -6223.843,E2 -6223.843} C_VEL
LIN {X 0,Y 497.802,Z 457.941,A -85,B 0,C 180,E1 -6224.251,E2 -6224.251} C_VEL
LIN {X 0,Y 498.045,Z 444.677,A -85,B 0,C 180,E1 -6224.505,E2 -6224.505} C_VEL
LIN {X 0,Y 498.448,Z 358.602,A -85,B 0,C 180,E1 -6225.754,E2 -6225.754} C_VEL
LIN {X 0,Y 496.245,Z 343.814,A -85,B 0,C 180,E1 -6226.045,E2 -6226.045} C_VEL
LIN {X 0,Y 496.852,Z 322.291,A -85,B 0,C 180,E1 -6229.414,E2 -6229.414} C_VEL
LIN {X 0,Y 497.47,Z 303.381,A -85,B 0,C 180,E1 -6232.422,E2 -6232.422} C_VEL
LIN {X 0,Y 497.681,Z 293.919,A -85,B 0,C 180,E1 -6233.953,E2 -6233.953} C_VEL
LIN {X 0,Y 495.763,Z 283.733,A -85,B 0,C 180,E1 -6235.73,E2 -6235.73} C_VEL
LIN {X 0,Y 495.742,Z 283.737,A -85,B 0,C 180,E1 -6238.816,E2 -6238.816} C_VEL
LIN {X 0,Y 495.753,Z 283.734,A -85,B 0,C 180,E1 -6241.724,E2 -6241.724} C_VEL
LIN {X 0,Y 495.76,Z 283.733,A -85,B 0,C 180,E1 -6244.692,E2 -6244.692} C_VEL
LIN {X 0,Y 495.719,Z 283.732,A -85,B 0,C 180,E1 -6247.562,E2 -6247.562} C_VEL
LIN {X 0,Y 495.763,Z 283.73,A -85,B 0,C 180,E1 -6250.7,E2 -6250.7} C_VEL
LIN {X 0,Y 495.725,Z 283.734,A -85,B 0,C 180,E1 -6254.001,E2 -6254.001} C_VEL
LIN {X 0,Y 495.723,Z 283.732,A -85,B 0,C 180,E1 -6257.116,E2 -6257.116} C_VEL
LIN {X 0,Y 495.756,Z 283.727,A -85,B 0,C 180,E1 -6259.953,E2 -6259.953} C_VEL
LIN {X 0,Y 495.725,Z 283.737,A -85,B 0,C 180,E1 -6262.553,E2 -6262.553} C_VEL
LIN {X 0,Y 495.768,Z 283.723,A -85,B 0,C 180,E1 -6265.456,E2 -6265.456} C_VEL
LIN {X 0,Y 495.752,Z 283.732,A -85,B 0,C 180,E1 -6268.364,E2 -6268.364} C_VEL
LIN {X 0,Y 495.784,Z 283.721,A -85,B 0,C 180,E1 -6271.507,E2 -6271.507} C_VEL
LIN {X 0,Y 495.777,Z 283.724,A -85,B 0,C 180,E1 -6273.931,E2 -6273.931} C_VEL
LIN {X 0,Y 495.755,Z 283.729,A -85,B 0,C 180,E1 -6277.139,E2 -6277.139} C_VEL
LIN {X 0,Y 495.775,Z 283.722,A -85,B 0,C 180,E1 -6280.11,E2 -6280.11} C_VEL
LIN {X 0,Y 495.785,Z 283.731,A -85,B 0,C 180,E1 -6282.681,E2 -6282.681} C_VEL
LIN {X 0,Y 495.787,Z 283.726,A -85,B 0,C 180,E1 -6285.217,E2 -6285.217} C_VEL
LIN {X 0,Y 495.848,Z 283.717,A -85,B 0,C 180,E1 -6288.555,E2 -6288.555} C_VEL
LIN {X 0,Y 495.87,Z 283.71,A -85,B 0,C 180,E1 -6291.852,E2 -6291.852} C_VEL
LIN {X 0,Y 495.892,Z 283.711,A -85,B 0,C 180,E1 -6294.307,E2 -6294.307} C_VEL
LIN {X 0,Y 495.991,Z 283.698,A -85,B 0,C 180,E1 -6297.564,E2 -6297.564} C_VEL
LIN {X 0,Y 495.996,Z 283.695,A -85,B 0,C 180,E1 -6300,E2 -6300} C_VEL
LIN {X 0,Y 495.991,Z 283.699,A -85,B 0,C 180,E1 -6302.437,E2 -6302.437} C_VEL
LIN {X 0,Y 495.892,Z 283.709,A -85,B 0,C 180,E1 -6305.694,E2 -6305.694} C_VEL
LIN {X 0,Y 495.87,Z 283.712,A -85,B 0,C 180,E1 -6308.148,E2 -6308.148} C_VEL
LIN {X 0,Y 495.849,Z 283.718,A -85,B 0,C 180,E1 -6311.446,E2 -6311.446} C_VEL
LIN {X 0,Y 495.787,Z 283.726,A -85,B 0,C 180,E1 -6314.783,E2 -6314.783} C_VEL
LIN {X 0,Y 495.763,Z 283.73,A -85,B 0,C 180,E1 -6317.32,E2 -6317.32} C_VEL
LIN {X 0,Y 495.768,Z 283.725,A -85,B 0,C 180,E1 -6319.891,E2 -6319.891} C_VEL
LIN {X 0,Y 495.756,Z 283.73,A -85,B 0,C 180,E1 -6322.861,E2 -6322.861} C_VEL
LIN {X 0,Y 495.777,Z 283.724,A -85,B 0,C 180,E1 -6326.069,E2 -6326.069} C_VEL
LIN {X 0,Y 495.767,Z 283.728,A -85,B 0,C 180,E1 -6328.816,E2 -6328.816} C_VEL
LIN {X 0,Y 495.752,Z 283.727,A -85,B 0,C 180,E1 -6331.726,E2 -6331.726} C_VEL
LIN {X 0,Y 495.762,Z 283.727,A -85,B 0,C 180,E1 -6334.694,E2 -6334.694} C_VEL
LIN {X 0,Y 495.727,Z 283.733,A -85,B 0,C 180,E1 -6337.562,E2 -6337.562} C_VEL
LIN {X 0,Y 495.748,Z 283.728,A -85,B 0,C 180,E1 -6340.702,E2 -6340.702} C_VEL
LIN {X 0,Y 495.722,Z 283.733,A -85,B 0,C 180,E1 -6344.003,E2 -6344.003} C_VEL
LIN {X 0,Y 495.703,Z 283.739,A -85,B 0,C 180,E1 -6347.115,E2 -6347.115} C_VEL
LIN {X 0,Y 495.742,Z 283.73,A -85,B 0,C 180,E1 -6350.361,E2 -6350.361} C_VEL
LIN {X 0,Y 495.71,Z 283.741,A -85,B 0,C 180,E1 -6353.455,E2 -6353.455} C_VEL
LIN {X 0,Y 495.752,Z 283.729,A -85,B 0,C 180,E1 -6356.436,E2 -6356.436} C_VEL
LIN {X 0,Y 495.745,Z 283.736,A -85,B 0,C 180,E1 -6359.313,E2 -6359.313} C_VEL
LIN {X 0,Y 495.748,Z 283.733,A -85,B 0,C 180,E1 -6360.757,E2 -6360.757} C_VEL
LIN {X 0,Y 495.463,Z 284.101,A -85,B 0,C 180,E1 -6361.205,E2 -6361.205} C_VEL
LIN {X 0,Y 494.254,Z 285.735,A -85,B 0,C 180,E1 -6361.845,E2 -6361.845} C_VEL
LIN {X 0,Y 492.589,Z 288.247,A -85,B 0,C 180,E1 -6362.442,E2 -6362.442} C_VEL
LIN {X 0,Y 490.391,Z 292.514,A -85,B 0,C 180,E1 -6363.221,E2 -6363.221} C_VEL
LIN {X 0,Y 489.434,Z 295.826,A -85,B 0,C 180,E1 -6363.81,E2 -6363.81} C_VEL
LIN {X 0,Y 489.348,Z 296.904,A -85,B 0,C 180,E1 -6364.012,E2 -6364.012} C_VEL
LIN {X 0,Y 489.303,Z 300.891,A -85,B 0,C 180,E1 -6364.763,E2 -6364.763} C_VEL
LIN {X 0,Y 491.891,Z 314.619,A -85,B 0,C 180,E1 -6365.065,E2 -6365.065} C_VEL
LIN {X 0,Y 491.18,Z 408.054,A -85,B 0,C 180,E1 -6366.458,E2 -6366.458} C_VEL
LIN {X 0,Y 491.024,Z 421.17,A -85,B 0,C 180,E1 -6366.822,E2 -6366.822} C_VEL
LIN {X 0,Y 490.672,Z 434.284,A -85,B 0,C 180,E1 -6367.361,E2 -6367.361} C_VEL
LIN {X 0,Y 490.339,Z 445.794,A -85,B 0,C 180,E1 -6368.01,E2 -6368.01} C_VEL
LIN {X 0,Y 489.894,Z 457.472,A -85,B 0,C 180,E1 -6368.859,E2 -6368.859} C_VEL
LIN {X 0,Y 489.454,Z 468.222,A -85,B 0,C 180,E1 -6369.842,E2 -6369.842} C_VEL
LIN {X 0,Y 489.078,Z 477.628,A -85,B 0,C 180,E1 -6370.919,E2 -6370.919} C_VEL
LIN {X 0,Y 488.736,Z 485.417,A -85,B 0,C 180,E1 -6372.006,E2 -6372.006} C_VEL
LIN {X 0,Y 488.482,Z 492.819,A -85,B 0,C 180,E1 -6373.277,E2 -6373.277} C_VEL
LIN {X 0,Y 488.249,Z 499.229,A -85,B 0,C 180,E1 -6374.672,E2 -6374.672} C_VEL
LIN {X 0,Y 488.118,Z 503.407,A -85,B 0,C 180,E1 -6375.832,E2 -6375.832} C_VEL
LIN {X 0,Y 488.039,Z 505.83,A -85,B 0,C 180,E1 -6376.679,E2 -6376.679} C_VEL
LIN {X 0,Y 487.992,Z 507.803,A -85,B 0,C 180,E1 -6377.525,E2 -6377.525} C_VEL
LIN {X 0,Y 487.97,Z 509.348,A -85,B 0,C 180,E1 -6378.368,E2 -6378.368} C_VEL
LIN {X 0,Y 487.909,Z 510.428,A -85,B 0,C 180,E1 -6379.208,E2 -6379.208} C_VEL
LIN {X 0,Y 487.861,Z 511.385,A -85,B 0,C 180,E1 -6380.883,E2 -6380.883} C_VEL
LIN {X 0,Y 487.918,Z 511.273,A -85,B 0,C 180,E1 -6381.719,E2 -6381.719} C_VEL
LIN {X 0,Y 487.988,Z 509.79,A -85,B 0,C 180,E1 -6383.384,E2 -6383.384} C_VEL
LIN {X 0,Y 488.026,Z 508.465,A -85,B 0,C 180,E1 -6384.215,E2 -6384.215} C_VEL
LIN {X 0,Y 488.012,Z 505.675,A -85,B 0,C 180,E1 -6385.458,E2 -6385.458} C_VEL
LIN {X 0,Y 488.196,Z 501.863,A -85,B 0,C 180,E1 -6386.699,E2 -6386.699} C_VEL
LIN {X 0,Y 488.263,Z 496.964,A -85,B 0,C 180,E1 -6387.938,E2 -6387.938} C_VEL
LIN {X 0,Y 488.569,Z 490.796,A -85,B 0,C 180,E1 -6389.176,E2 -6389.176} C_VEL
LIN {X 0,Y 488.806,Z 483.124,A -85,B 0,C 180,E1 -6390.412,E2 -6390.412} C_VEL
LIN {X 0,Y 489.2,Z 473.546,A -85,B 0,C 180,E1 -6391.647,E2 -6391.647} C_VEL
LIN {X 0,Y 489.523,Z 463.678,A -85,B 0,C 180,E1 -6392.675,E2 -6392.675} C_VEL
LIN {X 0,Y 489.919,Z 452.513,A -85,B 0,C 180,E1 -6393.599,E2 -6393.599} C_VEL
LIN {X 0,Y 490.392,Z 441.563,A -85,B 0,C 180,E1 -6394.316,E2 -6394.316} C_VEL
LIN {X 0,Y 490.61,Z 429.508,A -85,B 0,C 180,E1 -6394.931,E2 -6394.931} C_VEL
LIN {X 0,Y 490.883,Z 416.753,A -85,B 0,C 180,E1 -6395.392,E2 -6395.392} C_VEL
LIN {X 0,Y 491.171,Z 403.143,A -85,B 0,C 180,E1 -6395.697,E2 -6395.697} C_VEL
LIN {X 0,Y 491.77,Z 313.097,A -85,B 0,C 180,E1 -6397.019,E2 -6397.019} C_VEL
LIN {X 0,Y 489.27,Z 300.829,A -85,B 0,C 180,E1 -6397.291,E2 -6397.291} C_VEL
LIN {X 0,Y 489.384,Z 289.382,A -85,B 0,C 180,E1 -6399.506,E2 -6399.506} C_VEL
LIN {X 0,Y 488.698,Z 284.614,A -85,B 0,C 180,E1 -6400.514,E2 -6400.514} C_VEL
LIN {X 0,Y 488.743,Z 284.608,A -85,B 0,C 180,E1 -6402.457,E2 -6402.457} C_VEL
LIN {X 0,Y 488.764,Z 284.597,A -85,B 0,C 180,E1 -6405.856,E2 -6405.856} C_VEL
LIN {X 0,Y 488.733,Z 284.603,A -85,B 0,C 180,E1 -6409.314,E2 -6409.314} C_VEL
LIN {X 0,Y 488.702,Z 284.605,A -85,B 0,C 180,E1 -6411.957,E2 -6411.957} C_VEL
LIN {X 0,Y 488.702,Z 284.611,A -85,B 0,C 180,E1 -6415.04,E2 -6415.04} C_VEL
LIN {X 0,Y 488.698,Z 284.607,A -85,B 0,C 180,E1 -6418.332,E2 -6418.332} C_VEL
LIN {X 0,Y 488.687,Z 284.613,A -85,B 0,C 180,E1 -6421.181,E2 -6421.181} C_VEL
LIN {X 0,Y 488.724,Z 284.602,A -85,B 0,C 180,E1 -6424.114,E2 -6424.114} C_VEL
LIN {X 0,Y 488.675,Z 284.617,A -85,B 0,C 180,E1 -6427.16,E2 -6427.16} C_VEL
LIN {X 0,Y 488.699,Z 284.605,A -85,B 0,C 180,E1 -6430.341,E2 -6430.341} C_VEL
LIN {X 0,Y 488.678,Z 284.611,A -85,B 0,C 180,E1 -6433.656,E2 -6433.656} C_VEL
LIN {X 0,Y 488.678,Z 284.608,A -85,B 0,C 180,E1 -6436.344,E2 -6436.344} C_VEL
LIN {X 0,Y 488.709,Z 284.609,A -85,B 0,C 180,E1 -6439.674,E2 -6439.674} C_VEL
LIN {X 0,Y 488.665,Z 284.61,A -85,B 0,C 180,E1 -6442.839,E2 -6442.839} C_VEL
LIN {X 0,Y 488.723,Z 284.606,A -85,B 0,C 180,E1 -6445.886,E2 -6445.886} C_VEL
LIN {X 0,Y 488.695,Z 284.606,A -85,B 0,C 180,E1 -6448.82,E2 -6448.82} C_VEL
LIN {X 0,Y 488.713,Z 284.613,A -85,B 0,C 180,E1 -6451.669,E2 -6451.669} C_VEL
LIN {X 0,Y 488.701,Z 284.605,A -85,B 0,C 180,E1 -6454.96,E2 -6454.96} C_VEL
LIN {X 0,Y 488.702,Z 284.61,A -85,B 0,C 180,E1 -6458.043,E2 -6458.043} C_VEL
LIN {X 0,Y 488.74,Z 284.6,A -85,B 0,C 180,E1 -6460.686,E2 -6460.686} C_VEL
LIN {X 0,Y 488.762,Z 284.603,A -85,B 0,C 180,E1 -6464.145,E2 -6464.145} C_VEL
LIN {X 0,Y 488.742,Z 284.602,A -85,B 0,C 180,E1 -6467.543,E2 -6467.543} C_VEL
LIN {X 0,Y 488.742,Z 284.609,A -85,B 0,C 180,E1 -6470.063,E2 -6470.063} C_VEL
LIN {X 0,Y 488.824,Z 284.591,A -85,B 0,C 180,E1 -6472.769,E2 -6472.769} C_VEL
LIN {X 0,Y 488.793,Z 284.593,A -85,B 0,C 180,E1 -6475.051,E2 -6475.051} C_VEL
LIN {X 0,Y 488.945,Z 284.575,A -85,B 0,C 180,E1 -6477.528,E2 -6477.528} C_VEL
LIN {X 0,Y 488.945,Z 284.579,A -85,B 0,C 180,E1 -6480,E2 -6480} C_VEL
LIN {X 0,Y 488.944,Z 284.582,A -85,B 0,C 180,E1 -6482.471,E2 -6482.471} C_VEL
LIN {X 0,Y 488.815,Z 284.592,A -85,B 0,C 180,E1 -6485.776,E2 -6485.776} C_VEL
LIN {X 0,Y 488.758,Z 284.604,A -85,B 0,C 180,E1 -6488.267,E2 -6488.267} C_VEL
LIN {X 0,Y 488.787,Z 284.594,A -85,B 0,C 180,E1 -6491.613,E2 -6491.613} C_VEL
LIN {X 0,Y 488.758,Z 284.601,A -85,B 0,C 180,E1 -6495,E2 -6495} C_VEL
LIN {X 0,Y 488.747,Z 284.604,A -85,B 0,C 180,E1 -6498.442,E2 -6498.442} C_VEL
LIN {X 0,Y 488.71,Z 284.608,A -85,B 0,C 180,E1 -6501.071,E2 -6501.071} C_VEL
LIN {X 0,Y 488.672,Z 284.608,A -85,B 0,C 180,E1 -6503.746,E2 -6503.746} C_VEL
LIN {X 0,Y 488.699,Z 284.614,A -85,B 0,C 180,E1 -6506.921,E2 -6506.921} C_VEL
LIN {X 0,Y 488.707,Z 284.605,A -85,B 0,C 180,E1 -6510.22,E2 -6510.22} C_VEL
LIN {X 0,Y 488.713,Z 284.606,A -85,B 0,C 180,E1 -6513.479,E2 -6513.479} C_VEL
LIN {X 0,Y 488.676,Z 284.608,A -85,B 0,C 180,E1 -6516.353,E2 -6516.353} C_VEL
LIN {X 0,Y 488.695,Z 284.613,A -85,B 0,C 180,E1 -6519.255,E2 -6519.255} C_VEL
LIN {X 0,Y 488.669,Z 284.612,A -85,B 0,C 180,E1 -6521.594,E2 -6521.594} C_VEL
LIN {X 0,Y 488.704,Z 284.607,A -85,B 0,C 180,E1 -6524.802,E2 -6524.802} C_VEL
LIN {X 0,Y 488.652,Z 284.618,A -85,B 0,C 180,E1 -6527.47,E2 -6527.47} C_VEL
LIN {X 0,Y 488.706,Z 284.609,A -85,B 0,C 180,E1 -6529.673,E2 -6529.673} C_VEL
LIN {X 0,Y 488.663,Z 284.611,A -85,B 0,C 180,E1 -6532.839,E2 -6532.839} C_VEL
LIN {X 0,Y 488.721,Z 284.606,A -85,B 0,C 180,E1 -6535.886,E2 -6535.886} C_VEL
LIN {X 0,Y 488.693,Z 284.606,A -85,B 0,C 180,E1 -6538.82,E2 -6538.82} C_VEL
LIN {X 0,Y 488.711,Z 284.612,A -85,B 0,C 180,E1 -6541.669,E2 -6541.669} C_VEL
LIN {X 0,Y 488.746,Z 284.7,A -85,B 0,C 180,E1 -6544.187,E2 -6544.187} C_VEL
LIN {X 0,Y 490.672,Z 294.628,A -85,B 0,C 180,E1 -6545.907,E2 -6545.907} C_VEL
LIN {X 0,Y 490.352,Z 308.291,A -85,B 0,C 180,E1 -6548.121,E2 -6548.121} C_VEL
LIN {X 0,Y 489.711,Z 328.168,A -85,B 0,C 180,E1 -6551.296,E2 -6551.296} C_VEL
LIN {X 0,Y 489.242,Z 343.563,A -85,B 0,C 180,E1 -6553.733,E2 -6553.733} C_VEL
LIN {X 0,Y 491.649,Z 360.388,A -85,B 0,C 180,E1 -6554.064,E2 -6554.064} C_VEL
LIN {X 0,Y 491.039,Z 452.9,A -85,B 0,C 180,E1 -6555.441,E2 -6555.441} C_VEL
LIN {X 0,Y 490.695,Z 465.967,A -85,B 0,C 180,E1 -6555.801,E2 -6555.801} C_VEL
LIN {X 0,Y 490.357,Z 478.607,A -85,B 0,C 180,E1 -6556.32,E2 -6556.32} C_VEL
LIN {X 0,Y 489.971,Z 490.122,A -85,B 0,C 180,E1 -6556.961,E2 -6556.961} C_VEL
LIN {X 0,Y 489.54,Z 501.506,A -85,B 0,C 180,E1 -6557.774,E2 -6557.774} C_VEL
LIN {X 0,Y 489.147,Z 511.996,A -85,B 0,C 180,E1 -6558.71,E2 -6558.71} C_VEL
LIN {X 0,Y 488.799,Z 520.574,A -85,B 0,C 180,E1 -6559.646,E2 -6559.646} C_VEL
LIN {X 0,Y 488.494,Z 528.49,A -85,B 0,C 180,E1 -6560.685,E2 -6560.685} C_VEL
LIN {X 0,Y 488.257,Z 536.224,A -85,B 0,C 180,E1 -6561.932,E2 -6561.932} C_VEL
LIN {X 0,Y 488.073,Z 543.352,A -85,B 0,C 180,E1 -6563.385,E2 -6563.385} C_VEL
LIN {X 0,Y 488.018,Z 548.096,A -85,B 0,C 180,E1 -6564.628,E2 -6564.628} C_VEL
LIN {X 0,Y 487.932,Z 551.718,A -85,B 0,C 180,E1 -6565.87,E2 -6565.87} C_VEL
LIN {X 0,Y 487.965,Z 553.59,A -85,B 0,C 180,E1 -6566.697,E2 -6566.697} C_VEL
LIN {X 0,Y 487.932,Z 554.99,A -85,B 0,C 180,E1 -6567.523,E2 -6567.523} C_VEL
LIN {X 0,Y 487.892,Z 555.988,A -85,B 0,C 180,E1 -6568.349,E2 -6568.349} C_VEL
LIN {X 0,Y 487.825,Z 556.809,A -85,B 0,C 180,E1 -6569.999,E2 -6569.999} C_VEL
LIN {X 0,Y 487.892,Z 555.98,A -85,B 0,C 180,E1 -6571.65,E2 -6571.65} C_VEL
LIN {X 0,Y 487.932,Z 554.979,A -85,B 0,C 180,E1 -6572.476,E2 -6572.476} C_VEL
LIN {X 0,Y 487.969,Z 553.576,A -85,B 0,C 180,E1 -6573.302,E2 -6573.302} C_VEL
LIN {X 0,Y 487.921,Z 550.619,A -85,B 0,C 180,E1 -6574.543,E2 -6574.543} C_VEL
LIN {X 0,Y 488.02,Z 546.625,A -85,B 0,C 180,E1 -6575.785,E2 -6575.785} C_VEL
LIN {X 0,Y 488.18,Z 540.485,A -85,B 0,C 180,E1 -6577.236,E2 -6577.236} C_VEL
LIN {X 0,Y 488.346,Z 533.777,A -85,B 0,C 180,E1 -6578.482,E2 -6578.482} C_VEL
LIN {X 0,Y 488.608,Z 525.461,A -85,B 0,C 180,E1 -6579.73,E2 -6579.73} C_VEL
LIN {X 0,Y 488.972,Z 516.944,A -85,B 0,C 180,E1 -6580.768,E2 -6580.768} C_VEL
LIN {X 0,Y 489.407,Z 506.435,A -85,B 0,C 180,E1 -6581.807,E2 -6581.807} C_VEL
LIN {X 0,Y 489.815,Z 494.731,A -85,B 0,C 180,E1 -6582.736,E2 -6582.736} C_VEL
LIN {X 0,Y 490.216,Z 482.749,A -85,B 0,C 180,E1 -6583.471,E2 -6583.471} C_VEL
LIN {X 0,Y 490.597,Z 470.419,A -85,B 0,C 180,E1 -6584.042,E2 -6584.042} C_VEL
LIN {X 0,Y 490.942,Z 457.795,A -85,B 0,C 180,E1 -6584.455,E2 -6584.455} C_VEL
LIN {X 0,Y 491.185,Z 444.741,A -85,B 0,C 180,E1 -6584.712,E2 -6584.712} C_VEL
LIN {X 0,Y 491.567,Z 358.899,A -85,B 0,C 180,E1 -6585.98,E2 -6585.98} C_VEL
LIN {X 0,Y 489.246,Z 343.338,A -85,B 0,C 180,E1 -6586.309,E2 -6586.309} C_VEL
LIN {X 0,Y 489.876,Z 323.39,A -85,B 0,C 180,E1 -6589.484,E2 -6589.484} C_VEL
LIN {X 0,Y 490.539,Z 304.508,A -85,B 0,C 180,E1 -6592.535,E2 -6592.535} C_VEL
LIN {X 0,Y 490.751,Z 295.058,A -85,B 0,C 180,E1 -6594.088,E2 -6594.088} C_VEL
LIN {X 0,Y 488.718,Z 284.612,A -85,B 0,C 180,E1 -6595.957,E2 -6595.957} C_VEL
LIN {X 0,Y 488.708,Z 284.612,A -85,B 0,C 180,E1 -6599.271,E2 -6599.271} C_VEL
LIN {X 0,Y 488.701,Z 284.613,A -85,B 0,C 180,E1 -6602.147,E2 -6602.147} C_VEL
LIN {X 0,Y 488.712,Z 284.608,A -85,B 0,C 180,E1 -6605.115,E2 -6605.115} C_VEL
LIN {X 0,Y 488.673,Z 284.616,A -85,B 0,C 180,E1 -6608.2,E2 -6608.2} C_VEL
LIN {X 0,Y 488.716,Z 284.611,A -85,B 0,C 180,E1 -6610.344,E2 -6610.344} C_VEL
LIN {X 0,Y 488.682,Z 284.609,A -85,B 0,C 180,E1 -6613.654,E2 -6613.654} C_VEL
LIN {X 0,Y 488.682,Z 284.614,A -85,B 0,C 180,E1 -6616.345,E2 -6616.345} C_VEL
LIN {X 0,Y 488.73,Z 284.601,A -85,B 0,C 180,E1 -6619.676,E2 -6619.676} C_VEL
LIN {X 0,Y 488.676,Z 284.613,A -85,B 0,C 180,E1 -6622.841,E2 -6622.841} C_VEL
LIN {X 0,Y 488.721,Z 284.602,A -85,B 0,C 180,E1 -6625.886,E2 -6625.886} C_VEL
LIN {X 0,Y 488.689,Z 284.612,A -85,B 0,C 180,E1 -6628.82,E2 -6628.82} C_VEL
LIN {X 0,Y 488.741,Z 284.598,A -85,B 0,C 180,E1 -6631.671,E2 -6631.671} C_VEL
LIN {X 0,Y 488.723,Z 284.608,A -85,B 0,C 180,E1 -6634.443,E2 -6634.443} C_VEL
LIN {X 0,Y 488.718,Z 284.606,A -85,B 0,C 180,E1 -6637.153,E2 -6637.153} C_VEL
LIN {X 0,Y 488.725,Z 284.599,A -85,B 0,C 180,E1 -6639.811,E2 -6639.811} C_VEL
LIN {X 0,Y 488.732,Z 284.606,A -85,B 0,C 180,E1 -6642.423,E2 -6642.423} C_VEL
LIN {X 0,Y 488.759,Z 284.604,A -85,B 0,C 180,E1 -6645,E2 -6645} C_VEL
LIN {X 0,Y 488.802,Z 284.593,A -85,B 0,C 180,E1 -6648.388,E2 -6648.388} C_VEL
LIN {X 0,Y 488.814,Z 284.589,A -85,B 0,C 180,E1 -6651.734,E2 -6651.734} C_VEL
LIN {X 0,Y 488.851,Z 284.588,A -85,B 0,C 180,E1 -6654.224,E2 -6654.224} C_VEL
LIN {X 0,Y 488.959,Z 284.574,A -85,B 0,C 180,E1 -6657.529,E2 -6657.529} C_VEL
LIN {X 0,Y 488.951,Z 284.579,A -85,B 0,C 180,E1 -6660.824,E2 -6660.824} C_VEL
LIN {X 0,Y 488.958,Z 284.575,A -85,B 0,C 180,E1 -6662.472,E2 -6662.472} C_VEL
LIN {X 0,Y 488.851,Z 284.586,A -85,B 0,C 180,E1 -6665.776,E2 -6665.776} C_VEL
LIN {X 0,Y 488.815,Z 284.591,A -85,B 0,C 180,E1 -6668.267,E2 -6668.267} C_VEL
LIN {X 0,Y 488.803,Z 284.594,A -85,B 0,C 180,E1 -6671.613,E2 -6671.613} C_VEL
LIN {X 0,Y 488.759,Z 284.604,A -85,B 0,C 180,E1 -6675.001,E2 -6675.001} C_VEL
LIN {X 0,Y 488.744,Z 284.599,A -85,B 0,C 180,E1 -6678.443,E2 -6678.443} C_VEL
LIN {X 0,Y 488.704,Z 284.611,A -85,B 0,C 180,E1 -6681.071,E2 -6681.071} C_VEL
LIN {X 0,Y 488.673,Z 284.61,A -85,B 0,C 180,E1 -6683.747,E2 -6683.747} C_VEL
LIN {X 0,Y 488.789,Z 284.599,A -85,B 0,C 180,E1 -6686.944,E2 -6686.944} C_VEL
LIN {X 0,Y 488.706,Z 284.605,A -85,B 0,C 180,E1 -6690.363,E2 -6690.363} C_VEL
LIN {X 0,Y 488.728,Z 284.607,A -85,B 0,C 180,E1 -6693.484,E2 -6693.484} C_VEL
LIN {X 0,Y 488.681,Z 284.607,A -85,B 0,C 180,E1 -6696.355,E2 -6696.355} C_VEL
LIN {X 0,Y 488.695,Z 284.612,A -85,B 0,C 180,E1 -6699.255,E2 -6699.255} C_VEL
LIN {X 0,Y 488.695,Z 284.612,A -85,B 0,C 180,E1 -6701.599,E2 -6701.599} C_VEL
LIN {X 0,Y 488.7,Z 284.608,A -85,B 0,C 180,E1 -6704.803,E2 -6704.803} C_VEL
LIN {X 0,Y 488.666,Z 284.617,A -85,B 0,C 180,E1 -6707.472,E2 -6707.472} C_VEL
LIN {X 0,Y 488.687,Z 284.609,A -85,B 0,C 180,E1 -6710.745,E2 -6710.745} C_VEL
LIN {X 0,Y 488.666,Z 284.613,A -85,B 0,C 180,E1 -6713.868,E2 -6713.868} C_VEL
LIN {X 0,Y 488.736,Z 284.604,A -85,B 0,C 180,E1 -6716.878,E2 -6716.878} C_VEL
LIN {X 0,Y 488.718,Z 284.612,A -85,B 0,C 180,E1 -6719.781,E2 -6719.781} C_VEL
LIN {X 0,Y 488.778,Z 284.622,A -85,B 0,C 180,E1 -6721.628,E2 -6721.628} C_VEL
LIN {X 0,Y 489.4,Z 289.742,A -85,B 0,C 180,E1 -6722.644,E2 -6722.644} C_VEL
LIN {X 0,Y 489.348,Z 296.904,A -85,B 0,C 180,E1 -6724.012,E2 -6724.012} C_VEL
LIN {X 0,Y 488.997,Z 299.452,A -85,B 0,C 180,E1 -6724.336,E2 -6724.336} C_VEL
LIN {X 0,Y 488.227,Z 302.688,A -85,B 0,C 180,E1 -6724.56,E2 -6724.56} C_VEL
LIN {X 0,Y 486.817,Z 308.237,A -85,B 0,C 180,E1 -6724.757,E2 -6724.757} C_VEL
LIN {X 0,Y 484.907,Z 319.124,A -85,B 0,C 180,E1 -6724.875,E2 -6724.875} C_VEL
LIN {X 0,Y 485.01,Z 327.108,A -85,B 0,C 180,E1 -6725.002,E2 -6725.002} C_VEL
LIN {X 0,Y 484.366,Z 408.698,A -85,B 0,C 180,E1 -6726.242,E2 -6726.242} C_VEL
LIN {X 0,Y 484.173,Z 422.241,A -85,B 0,C 180,E1 -6726.629,E2 -6726.629} C_VEL
LIN {X 0,Y 483.823,Z 434.296,A -85,B 0,C 180,E1 -6727.135,E2 -6727.135} C_VEL
LIN {X 0,Y 483.469,Z 445.894,A -85,B 0,C 180,E1 -6727.794,E2 -6727.794} C_VEL
LIN {X 0,Y 482.994,Z 457.776,A -85,B 0,C 180,E1 -6728.669,E2 -6728.669} C_VEL
LIN {X 0,Y 482.529,Z 468.389,A -85,B 0,C 180,E1 -6729.652,E2 -6729.652} C_VEL
LIN {X 0,Y 482.179,Z 476.989,A -85,B 0,C 180,E1 -6730.635,E2 -6730.635} C_VEL
LIN {X 0,Y 481.752,Z 485.363,A -85,B 0,C 180,E1 -6731.804,E2 -6731.804} C_VEL
LIN {X 0,Y 481.483,Z 492.479,A -85,B 0,C 180,E1 -6733.027,E2 -6733.027} C_VEL
LIN {X 0,Y 481.222,Z 498.433,A -85,B 0,C 180,E1 -6734.296,E2 -6734.296} C_VEL
LIN {X 0,Y 481.061,Z 503.316,A -85,B 0,C 180,E1 -6735.62,E2 -6735.62} C_VEL
LIN {X 0,Y 480.935,Z 506.915,A -85,B 0,C 180,E1 -6736.909,E2 -6736.909} C_VEL
LIN {X 0,Y 480.888,Z 509.626,A -85,B 0,C 180,E1 -6738.291,E2 -6738.291} C_VEL
LIN {X 0,Y 480.789,Z 511.359,A -85,B 0,C 180,E1 -6739.898,E2 -6739.898} C_VEL
LIN {X 0,Y 480.815,Z 511.636,A -85,B 0,C 180,E1 -6741.596,E2 -6741.596} C_VEL
LIN {X 0,Y 480.842,Z 511.178,A -85,B 0,C 180,E1 -6742.442,E2 -6742.442} C_VEL
LIN {X 0,Y 480.942,Z 509.011,A -85,B 0,C 180,E1 -6744.129,E2 -6744.129} C_VEL
LIN {X 0,Y 480.913,Z 506.322,A -85,B 0,C 180,E1 -6745.39,E2 -6745.39} C_VEL
LIN {X 0,Y 481.105,Z 502.616,A -85,B 0,C 180,E1 -6746.651,E2 -6746.651} C_VEL
LIN {X 0,Y 481.201,Z 497.823,A -85,B 0,C 180,E1 -6747.908,E2 -6747.908} C_VEL
LIN {X 0,Y 481.484,Z 491.777,A -85,B 0,C 180,E1 -6749.164,E2 -6749.164} C_VEL
LIN {X 0,Y 481.766,Z 484.292,A -85,B 0,C 180,E1 -6750.418,E2 -6750.418} C_VEL
LIN {X 0,Y 482.09,Z 476.645,A -85,B 0,C 180,E1 -6751.462,E2 -6751.462} C_VEL
LIN {X 0,Y 482.496,Z 466.285,A -85,B 0,C 180,E1 -6752.609,E2 -6752.609} C_VEL
LIN {X 0,Y 482.87,Z 455.769,A -85,B 0,C 180,E1 -6753.547,E2 -6753.547} C_VEL
LIN {X 0,Y 483.302,Z 445.581,A -85,B 0,C 180,E1 -6754.275,E2 -6754.275} C_VEL
LIN {X 0,Y 483.655,Z 434.568,A -85,B 0,C 180,E1 -6754.898,E2 -6754.898} C_VEL
LIN {X 0,Y 483.908,Z 421.529,A -85,B 0,C 180,E1 -6755.444,E2 -6755.444} C_VEL
LIN {X 0,Y 484.2,Z 408.5,A -85,B 0,C 180,E1 -6755.806,E2 -6755.806} C_VEL
LIN {X 0,Y 484.906,Z 313.924,A -85,B 0,C 180,E1 -6757.23,E2 -6757.23} C_VEL
LIN {X 0,Y 482.331,Z 301.003,A -85,B 0,C 180,E1 -6757.536,E2 -6757.536} C_VEL
LIN {X 0,Y 482.388,Z 290.178,A -85,B 0,C 180,E1 -6759.646,E2 -6759.646} C_VEL
LIN {X 0,Y 481.668,Z 285.49,A -85,B 0,C 180,E1 -6760.616,E2 -6760.616} C_VEL
LIN {X 0,Y 481.687,Z 285.486,A -85,B 0,C 180,E1 -6762.642,E2 -6762.642} C_VEL
LIN {X 0,Y 481.73,Z 285.473,A -85,B 0,C 180,E1 -6765.658,E2 -6765.658} C_VEL
LIN {X 0,Y 481.71,Z 285.485,A -85,B 0,C 180,E1 -6768.722,E2 -6768.722} C_VEL
LIN {X 0,Y 481.651,Z 285.484,A -85,B 0,C 180,E1 -6771.395,E2 -6771.395} C_VEL
LIN {X 0,Y 481.653,Z 285.483,A -85,B 0,C 180,E1 -6774.115,E2 -6774.115} C_VEL
LIN {X 0,Y 481.656,Z 285.488,A -85,B 0,C 180,E1 -6777.117,E2 -6777.117} C_VEL
LIN {X 0,Y 481.66,Z 285.482,A -85,B 0,C 180,E1 -6779.743,E2 -6779.743} C_VEL
LIN {X 0,Y 481.657,Z 285.486,A -85,B 0,C 180,E1 -6782.676,E2 -6782.676} C_VEL
LIN {X 0,Y 481.636,Z 285.486,A -85,B 0,C 180,E1 -6785.71,E2 -6785.71} C_VEL
LIN {X 0,Y 481.671,Z 285.485,A -85,B 0,C 180,E1 -6788.86,E2 -6788.86} C_VEL
LIN {X 0,Y 481.62,Z 285.487,A -85,B 0,C 180,E1 -6792.164,E2 -6792.164} C_VEL
LIN {X 0,Y 481.659,Z 285.482,A -85,B 0,C 180,E1 -6794.458,E2 -6794.458} C_VEL
LIN {X 0,Y 481.62,Z 285.489,A -85,B 0,C 180,E1 -6796.855,E2 -6796.855} C_VEL
LIN {X 0,Y 481.66,Z 285.483,A -85,B 0,C 180,E1 -6800.057,E2 -6800.057} C_VEL
LIN {X 0,Y 481.623,Z 285.494,A -85,B 0,C 180,E1 -6803.378,E2 -6803.378} C_VEL
LIN {X 0,Y 481.675,Z 285.48,A -85,B 0,C 180,E1 -6806.327,E2 -6806.327} C_VEL
LIN {X 0,Y 481.654,Z 285.489,A -85,B 0,C 180,E1 -6809.418,E2 -6809.418} C_VEL
LIN {X 0,Y 481.663,Z 285.484,A -85,B 0,C 180,E1 -6812.165,E2 -6812.165} C_VEL
LIN {X 0,Y 481.675,Z 285.48,A -85,B 0,C 180,E1 -6814.967,E2 -6814.967} C_VEL
LIN {X 0,Y 481.653,Z 285.49,A -85,B 0,C 180,E1 -6817.705,E2 -6817.705} C_VEL
LIN {X 0,Y 481.704,Z 285.478,A -85,B 0,C 180,E1 -6820.393,E2 -6820.393} C_VEL
LIN {X 0,Y 481.669,Z 285.481,A -85,B 0,C 180,E1 -6823.033,E2 -6823.033} C_VEL
LIN {X 0,Y 481.685,Z 285.483,A -85,B 0,C 180,E1 -6825.638,E2 -6825.638} C_VEL
LIN {X 0,Y 481.739,Z 285.478,A -85,B 0,C 180,E1 -6828.215,E2 -6828.215} C_VEL
LIN {X 0,Y 481.724,Z 285.476,A -85,B 0,C 180,E1 -6831.611,E2 -6831.611} C_VEL
LIN {X 0,Y 481.779,Z 285.476,A -85,B 0,C 180,E1 -6834.139,E2 -6834.139} C_VEL
LIN {X 0,Y 481.911,Z 285.451,A -85,B 0,C 180,E1 -6837.492,E2 -6837.492} C_VEL
LIN {X 0,Y 481.914,Z 285.455,A -85,B 0,C 180,E1 -6840,E2 -6840} C_VEL
LIN {X 0,Y 481.91,Z 285.457,A -85,B 0,C 180,E1 -6842.507,E2 -6842.507} C_VEL
LIN {X 0,Y 481.777,Z 285.469,A -85,B 0,C 180,E1 -6845.861,E2 -6845.861} C_VEL
LIN {X 0,Y 481.716,Z 285.483,A -85,B 0,C 180,E1 -6848.389,E2 -6848.389} C_VEL
LIN {X 0,Y 481.738,Z 285.473,A -85,B 0,C 180,E1 -6851.785,E2 -6851.785} C_VEL
LIN {X 0,Y 481.742,Z 285.473,A -85,B 0,C 180,E1 -6855.224,E2 -6855.224} C_VEL
LIN {X 0,Y 481.707,Z 285.485,A -85,B 0,C 180,E1 -6858.722,E2 -6858.722} C_VEL
LIN {X 0,Y 481.648,Z 285.485,A -85,B 0,C 180,E1 -6861.395,E2 -6861.395} C_VEL
LIN {X 0,Y 481.65,Z 285.484,A -85,B 0,C 180,E1 -6864.114,E2 -6864.114} C_VEL
LIN {X 0,Y 481.654,Z 285.488,A -85,B 0,C 180,E1 -6867.116,E2 -6867.116} C_VEL
LIN {X 0,Y 481.658,Z 285.482,A -85,B 0,C 180,E1 -6869.743,E2 -6869.743} C_VEL
LIN {X 0,Y 481.654,Z 285.487,A -85,B 0,C 180,E1 -6872.676,E2 -6872.676} C_VEL
LIN {X 0,Y 481.634,Z 285.486,A -85,B 0,C 180,E1 -6875.71,E2 -6875.71} C_VEL
LIN {X 0,Y 481.668,Z 285.486,A -85,B 0,C 180,E1 -6878.859,E2 -6878.859} C_VEL
LIN {X 0,Y 481.618,Z 285.487,A -85,B 0,C 180,E1 -6882.164,E2 -6882.164} C_VEL
LIN {X 0,Y 481.656,Z 285.483,A -85,B 0,C 180,E1 -6884.458,E2 -6884.458} C_VEL
LIN {X 0,Y 481.618,Z 285.49,A -85,B 0,C 180,E1 -6886.855,E2 -6886.855} C_VEL
LIN {X 0,Y 481.658,Z 285.483,A -85,B 0,C 180,E1 -6890.057,E2 -6890.057} C_VEL
LIN {X 0,Y 481.62,Z 285.495,A -85,B 0,C 180,E1 -6893.378,E2 -6893.378} C_VEL
LIN {X 0,Y 481.673,Z 285.481,A -85,B 0,C 180,E1 -6896.327,E2 -6896.327} C_VEL
LIN {X 0,Y 481.652,Z 285.489,A -85,B 0,C 180,E1 -6899.418,E2 -6899.418} C_VEL
LIN {X 0,Y 481.661,Z 285.486,A -85,B 0,C 180,E1 -6902.165,E2 -6902.165} C_VEL
LIN {X 0,Y 481.685,Z 285.569,A -85,B 0,C 180,E1 -6904.012,E2 -6904.012} C_VEL
LIN {X 0,Y 483.8,Z 296.896,A -85,B 0,C 180,E1 -6905.999,E2 -6905.999} C_VEL
LIN {X 0,Y 483.185,Z 314.651,A -85,B 0,C 180,E1 -6908.9,E2 -6908.9} C_VEL
LIN {X 0,Y 482.592,Z 332.315,A -85,B 0,C 180,E1 -6911.753,E2 -6911.753} C_VEL
LIN {X 0,Y 482.231,Z 343.337,A -85,B 0,C 180,E1 -6913.51,E2 -6913.51} C_VEL
LIN {X 0,Y 484.799,Z 361.281,A -85,B 0,C 180,E1 -6913.863,E2 -6913.863} C_VEL
LIN {X 0,Y 484.156,Z 452.142,A -85,B 0,C 180,E1 -6915.23,E2 -6915.23} C_VEL
LIN {X 0,Y 483.836,Z 465.362,A -85,B 0,C 180,E1 -6915.596,E2 -6915.596} C_VEL
LIN {X 0,Y 483.41,Z 478.08,A -85,B 0,C 180,E1 -6916.12,E2 -6916.12} C_VEL
LIN {X 0,Y 483.016,Z 489.388,A -85,B 0,C 180,E1 -6916.752,E2 -6916.752} C_VEL
LIN {X 0,Y 482.57,Z 501.079,A -85,B 0,C 180,E1 -6917.595,E2 -6917.595} C_VEL
LIN {X 0,Y 482.167,Z 511.601,A -85,B 0,C 180,E1 -6918.545,E2 -6918.545} C_VEL
LIN {X 0,Y 481.754,Z 520.194,A -85,B 0,C 180,E1 -6919.493,E2 -6919.493} C_VEL
LIN {X 0,Y 481.458,Z 528.126,A -85,B 0,C 180,E1 -6920.548,E2 -6920.548} C_VEL
LIN {X 0,Y 481.184,Z 535.873,A -85,B 0,C 180,E1 -6921.812,E2 -6921.812} C_VEL
LIN {X 0,Y 480.976,Z 543.009,A -85,B 0,C 180,E1 -6923.286,E2 -6923.286} C_VEL
LIN {X 0,Y 480.93,Z 547.76,A -85,B 0,C 180,E1 -6924.549,E2 -6924.549} C_VEL
LIN {X 0,Y 480.831,Z 551.384,A -85,B 0,C 180,E1 -6925.808,E2 -6925.808} C_VEL
LIN {X 0,Y 480.889,Z 553.258,A -85,B 0,C 180,E1 -6926.648,E2 -6926.648} C_VEL
LIN {X 0,Y 480.844,Z 554.659,A -85,B 0,C 180,E1 -6927.486,E2 -6927.486} C_VEL
LIN {X 0,Y 480.823,Z 555.658,A -85,B 0,C 180,E1 -6928.324,E2 -6928.324} C_VEL
LIN {X 0,Y 480.749,Z 556.48,A -85,B 0,C 180,E1 -6929.999,E2 -6929.999} C_VEL
LIN {X 0,Y 480.823,Z 555.652,A -85,B 0,C 180,E1 -6931.675,E2 -6931.675} C_VEL
LIN {X 0,Y 480.845,Z 554.65,A -85,B 0,C 180,E1 -6932.513,E2 -6932.513} C_VEL
LIN {X 0,Y 480.893,Z 553.247,A -85,B 0,C 180,E1 -6933.351,E2 -6933.351} C_VEL
LIN {X 0,Y 480.839,Z 550.29,A -85,B 0,C 180,E1 -6934.61,E2 -6934.61} C_VEL
LIN {X 0,Y 480.923,Z 546.299,A -85,B 0,C 180,E1 -6935.871,E2 -6935.871} C_VEL
LIN {X 0,Y 481.105,Z 540.167,A -85,B 0,C 180,E1 -6937.343,E2 -6937.343} C_VEL
LIN {X 0,Y 481.291,Z 533.468,A -85,B 0,C 180,E1 -6938.608,E2 -6938.608} C_VEL
LIN {X 0,Y 481.561,Z 525.162,A -85,B 0,C 180,E1 -6939.873,E2 -6939.873} C_VEL
LIN {X 0,Y 481.977,Z 516.67,A -85,B 0,C 180,E1 -6940.927,E2 -6940.927} C_VEL
LIN {X 0,Y 482.406,Z 506.202,A -85,B 0,C 180,E1 -6941.98,E2 -6941.98} C_VEL
LIN {X 0,Y 482.86,Z 494.899,A -85,B 0,C 180,E1 -6942.893,E2 -6942.893} C_VEL
LIN {X 0,Y 483.295,Z 482.592,A -85,B 0,C 180,E1 -6943.668,E2 -6943.668} C_VEL
LIN {X 0,Y 483.724,Z 470.335,A -85,B 0,C 180,E1 -6944.245,E2 -6944.245} C_VEL
LIN {X 0,Y 484.106,Z 456.907,A -85,B 0,C 180,E1 -6944.69,E2 -6944.69} C_VEL
LIN {X 0,Y 484.382,Z 443.391,A -85,B 0,C 180,E1 -6944.95,E2 -6944.95} C_VEL
LIN {X 0,Y 484.835,Z 360.136,A -85,B 0,C 180,E1 -6946.197,E2 -6946.197} C_VEL
LIN {X 0,Y 482.242,Z 343.018,A -85,B 0,C 180,E1 -6946.564,E2 -6946.564} C_VEL
LIN {X 0,Y 482.889,Z 324.511,A -85,B 0,C 180,E1 -6949.556,E2 -6949.556} C_VEL
LIN {X 0,Y 483.609,Z 305.652,A -85,B 0,C 180,E1 -6952.65,E2 -6952.65} C_VEL
LIN {X 0,Y 483.791,Z 296.213,A -85,B 0,C 180,E1 -6954.228,E2 -6954.228} C_VEL
LIN {X 0,Y 481.654,Z 285.492,A -85,B 0,C 180,E1 -6956.192,E2 -6956.192} C_VEL
LIN {X 0,Y 481.652,Z 285.493,A -85,B 0,C 180,E1 -6958.897,E2 -6958.897} C_VEL
LIN {X 0,Y 481.655,Z 285.491,A -85,B 0,C 180,E1 -6962.188,E2 -6962.188} C_VEL
LIN {X 0,Y 481.657,Z 285.487,A -85,B 0,C 180,E1 -6965.203,E2 -6965.203} C_VEL
LIN {X 0,Y 481.666,Z 285.484,A -85,B 0,C 180,E1 -6968.859,E2 -6968.859} C_VEL
LIN {X 0,Y 481.65,Z 285.485,A -85,B 0,C 180,E1 -6971.912,E2 -6971.912} C_VEL
LIN {X 0,Y 481.652,Z 285.492,A -85,B 0,C 180,E1 -6974.457,E2 -6974.457} C_VEL
LIN {X 0,Y 481.645,Z 285.486,A -85,B 0,C 180,E1 -6977.839,E2 -6977.839} C_VEL
LIN {X 0,Y 481.678,Z 285.487,A -85,B 0,C 180,E1 -6980.651,E2 -6980.651} C_VEL
LIN {X 0,Y 481.624,Z 285.487,A -85,B 0,C 180,E1 -6983.376,E2 -6983.376} C_VEL
LIN {X 0,Y 481.673,Z 285.484,A -85,B 0,C 180,E1 -6986.327,E2 -6986.327} C_VEL
LIN {X 0,Y 481.647,Z 285.483,A -85,B 0,C 180,E1 -6989.417,E2 -6989.417} C_VEL
LIN {X 0,Y 481.696,Z 285.478,A -85,B 0,C 180,E1 -6992.168,E2 -6992.168} C_VEL
LIN {X 0,Y 481.689,Z 285.48,A -85,B 0,C 180,E1 -6994.968,E2 -6994.968} C_VEL
LIN {X 0,Y 481.645,Z 285.484,A -85,B 0,C 180,E1 -6997.705,E2 -6997.705} C_VEL
LIN {X 0,Y 481.705,Z 285.477,A -85,B 0,C 180,E1 -7000.393,E2 -7000.393} C_VEL
LIN {X 0,Y 481.688,Z 285.481,A -85,B 0,C 180,E1 -7003.034,E2 -7003.034} C_VEL
LIN {X 0,Y 481.687,Z 285.48,A -85,B 0,C 180,E1 -7005.639,E2 -7005.639} C_VEL
LIN {X 0,Y 481.747,Z 285.47,A -85,B 0,C 180,E1 -7008.215,E2 -7008.215} C_VEL
LIN {X 0,Y 481.759,Z 285.468,A -85,B 0,C 180,E1 -7011.612,E2 -7011.612} C_VEL
LIN {X 0,Y 481.812,Z 285.464,A -85,B 0,C 180,E1 -7014.14,E2 -7014.14} C_VEL
LIN {X 0,Y 481.926,Z 285.451,A -85,B 0,C 180,E1 -7017.493,E2 -7017.493} C_VEL
LIN {X 0,Y 481.902,Z 285.456,A -85,B 0,C 180,E1 -7020.836,E2 -7020.836} C_VEL
LIN {X 0,Y 481.925,Z 285.452,A -85,B 0,C 180,E1 -7022.508,E2 -7022.508} C_VEL
LIN {X 0,Y 481.813,Z 285.462,A -85,B 0,C 180,E1 -7025.861,E2 -7025.861} C_VEL
LIN {X 0,Y 481.76,Z 285.47,A -85,B 0,C 180,E1 -7028.389,E2 -7028.389} C_VEL
LIN {X 0,Y 481.748,Z 285.472,A -85,B 0,C 180,E1 -7031.785,E2 -7031.785} C_VEL
LIN {X 0,Y 481.74,Z 285.479,A -85,B 0,C 180,E1 -7035.225,E2 -7035.225} C_VEL
LIN {X 0,Y 481.706,Z 285.479,A -85,B 0,C 180,E1 -7038.722,E2 -7038.722} C_VEL
LIN {X 0,Y 481.643,Z 285.489,A -85,B 0,C 180,E1 -7041.395,E2 -7041.395} C_VEL
LIN {X 0,Y 481.655,Z 285.483,A -85,B 0,C 180,E1 -7044.115,E2 -7044.115} C_VEL
LIN {X 0,Y 481.744,Z 285.48,A -85,B 0,C 180,E1 -7047.139,E2 -7047.139} C_VEL
LIN {X 0,Y 481.676,Z 285.483,A -85,B 0,C 180,E1 -7049.742,E2 -7049.742} C_VEL
LIN {X 0,Y 481.668,Z 285.48,A -85,B 0,C 180,E1 -7052.675,E2 -7052.675} C_VEL
LIN {X 0,Y 481.635,Z 285.488,A -85,B 0,C 180,E1 -7055.71,E2 -7055.71} C_VEL
LIN {X 0,Y 481.667,Z 285.482,A -85,B 0,C 180,E1 -7058.86,E2 -7058.86} C_VEL
LIN {X 0,Y 481.64,Z 285.487,A -85,B 0,C 180,E1 -7061.912,E2 -7061.912} C_VEL
LIN {X 0,Y 481.653,Z 285.484,A -85,B 0,C 180,E1 -7064.459,E2 -7064.459} C_VEL
LIN {X 0,Y 481.626,Z 285.491,A -85,B 0,C 180,E1 -7067.838,E2 -7067.838} C_VEL
LIN {X 0,Y 481.656,Z 285.489,A -85,B 0,C 180,E1 -7071.14,E2 -7071.14} C_VEL
LIN {X 0,Y 481.658,Z 285.483,A -85,B 0,C 180,E1 -7074.798,E2 -7074.798} C_VEL
LIN {X 0,Y 481.655,Z 285.49,A -85,B 0,C 180,E1 -7077.812,E2 -7077.812} C_VEL
LIN {X 0,Y 481.721,Z 285.486,A -85,B 0,C 180,E1 -7081.429,E2 -7081.429} C_VEL
LIN {X 0,Y 482.478,Z 290.822,A -85,B 0,C 180,E1 -7082.517,E2 -7082.517} C_VEL
LIN {X 0,Y 482.363,Z 301.113,A -85,B 0,C 180,E1 -7084.498,E2 -7084.498} C_VEL
LIN {X 0,Y 485.115,Z 315.408,A -85,B 0,C 180,E1 -7084.827,E2 -7084.827} C_VEL
LIN {X 0,Y 485.01,Z 327.108,A -85,B 0,C 180,E1 -7085.002,E2 -7085.002} C_VEL
LIN {X 0,Y 484.38,Z 332.953,A -85,B 0,C 180,E1 -7085.067,E2 -7085.067} C_VEL
LIN {X 0,Y 478.661,Z 351.956,A -85,B 0,C 180,E1 -7085.145,E2 -7085.145} C_VEL
LIN {X 0,Y 477.964,Z 357.805,A -85,B 0,C 180,E1 -7085.209,E2 -7085.209} C_VEL
LIN {X 0,Y 477.546,Z 409.707,A -85,B 0,C 180,E1 -7086.025,E2 -7086.025} C_VEL
LIN {X 0,Y 477.337,Z 423.552,A -85,B 0,C 180,E1 -7086.436,E2 -7086.436} C_VEL
LIN {X 0,Y 476.946,Z 435.519,A -85,B 0,C 180,E1 -7086.958,E2 -7086.958} C_VEL
LIN {X 0,Y 476.52,Z 447.68,A -85,B 0,C 180,E1 -7087.681,E2 -7087.681} C_VEL
LIN {X 0,Y 476.036,Z 459.237,A -85,B 0,C 180,E1 -7088.564,E2 -7088.564} C_VEL
LIN {X 0,Y 475.56,Z 469.623,A -85,B 0,C 180,E1 -7089.566,E2 -7089.566} C_VEL
LIN {X 0,Y 475.091,Z 479.717,A -85,B 0,C 180,E1 -7090.784,E2 -7090.784} C_VEL
LIN {X 0,Y 474.671,Z 488.494,A -85,B 0,C 180,E1 -7092.108,E2 -7092.108} C_VEL
LIN {X 0,Y 474.336,Z 495.443,A -85,B 0,C 180,E1 -7093.429,E2 -7093.429} C_VEL
LIN {X 0,Y 474.074,Z 501.771,A -85,B 0,C 180,E1 -7094.964,E2 -7094.964} C_VEL
LIN {X 0,Y 473.914,Z 505.849,A -85,B 0,C 180,E1 -7096.275,E2 -7096.275} C_VEL
LIN {X 0,Y 473.86,Z 507.935,A -85,B 0,C 180,E1 -7097.146,E2 -7097.146} C_VEL
LIN {X 0,Y 473.82,Z 509.936,A -85,B 0,C 180,E1 -7098.227,E2 -7098.227} C_VEL
LIN {X 0,Y 473.708,Z 511.62,A -85,B 0,C 180,E1 -7099.745,E2 -7099.745} C_VEL
LIN {X 0,Y 473.728,Z 511.99,A -85,B 0,C 180,E1 -7101.469,E2 -7101.469} C_VEL
LIN {X 0,Y 473.752,Z 511.597,A -85,B 0,C 180,E1 -7102.328,E2 -7102.328} C_VEL
LIN {X 0,Y 473.836,Z 510.239,A -85,B 0,C 180,E1 -7103.598,E2 -7103.598} C_VEL
LIN {X 0,Y 473.82,Z 506.958,A -85,B 0,C 180,E1 -7105.321,E2 -7105.321} C_VEL
LIN {X 0,Y 474.018,Z 503.351,A -85,B 0,C 180,E1 -7106.601,E2 -7106.601} C_VEL
LIN {X 0,Y 474.14,Z 498.663,A -85,B 0,C 180,E1 -7107.877,E2 -7107.877} C_VEL
LIN {X 0,Y 474.48,Z 491.629,A -85,B 0,C 180,E1 -7109.364,E2 -7109.364} C_VEL
LIN {X 0,Y 474.785,Z 484.003,A -85,B 0,C 180,E1 -7110.637,E2 -7110.637} C_VEL
LIN {X 0,Y 475.201,Z 474.461,A -85,B 0,C 180,E1 -7111.907,E2 -7111.907} C_VEL
LIN {X 0,Y 475.564,Z 464.644,A -85,B 0,C 180,E1 -7112.965,E2 -7112.965} C_VEL
LIN {X 0,Y 476.026,Z 453.545,A -85,B 0,C 180,E1 -7113.916,E2 -7113.916} C_VEL
LIN {X 0,Y 476.553,Z 442.66,A -85,B 0,C 180,E1 -7114.653,E2 -7114.653} C_VEL
LIN {X 0,Y 476.795,Z 430.718,A -85,B 0,C 180,E1 -7115.286,E2 -7115.286} C_VEL
LIN {X 0,Y 477.102,Z 418.284,A -85,B 0,C 180,E1 -7115.76,E2 -7115.76} C_VEL
LIN {X 0,Y 477.392,Z 405.245,A -85,B 0,C 180,E1 -7116.074,E2 -7116.074} C_VEL
LIN {X 0,Y 478.085,Z 314.964,A -85,B 0,C 180,E1 -7117.439,E2 -7117.439} C_VEL
LIN {X 0,Y 475.382,Z 301.281,A -85,B 0,C 180,E1 -7117.764,E2 -7117.764} C_VEL
LIN {X 0,Y 475.439,Z 292.063,A -85,B 0,C 180,E1 -7119.573,E2 -7119.573} C_VEL
LIN {X 0,Y 474.65,Z 286.364,A -85,B 0,C 180,E1 -7120.774,E2 -7120.774} C_VEL
LIN {X 0,Y 474.647,Z 286.362,A -85,B 0,C 180,E1 -7122.833,E2 -7122.833} C_VEL
LIN {X 0,Y 474.686,Z 286.351,A -85,B 0,C 180,E1 -7125.767,E2 -7125.767} C_VEL
LIN {X 0,Y 474.663,Z 286.358,A -85,B 0,C 180,E1 -7129.011,E2 -7129.011} C_VEL
LIN {X 0,Y 474.593,Z 286.362,A -85,B 0,C 180,E1 -7131.729,E2 -7131.729} C_VEL
LIN {X 0,Y 474.63,Z 286.361,A -85,B 0,C 180,E1 -7134.495,E2 -7134.495} C_VEL
LIN {X 0,Y 474.603,Z 286.364,A -85,B 0,C 180,E1 -7137.327,E2 -7137.327} C_VEL
LIN {X 0,Y 474.591,Z 286.363,A -85,B 0,C 180,E1 -7140.232,E2 -7140.232} C_VEL
LIN {X 0,Y 474.62,Z 286.365,A -85,B 0,C 180,E1 -7143.222,E2 -7143.222} C_VEL
LIN {X 0,Y 474.589,Z 286.363,A -85,B 0,C 180,E1 -7146.324,E2 -7146.324} C_VEL
LIN {X 0,Y 474.627,Z 286.362,A -85,B 0,C 180,E1 -7149.548,E2 -7149.548} C_VEL
LIN {X 0,Y 474.581,Z 286.364,A -85,B 0,C 180,E1 -7152.23,E2 -7152.23} C_VEL
LIN {X 0,Y 474.621,Z 286.368,A -85,B 0,C 180,E1 -7155.298,E2 -7155.298} C_VEL
LIN {X 0,Y 474.597,Z 286.362,A -85,B 0,C 180,E1 -7158.211,E2 -7158.211} C_VEL
LIN {X 0,Y 474.604,Z 286.369,A -85,B 0,C 180,E1 -7161.541,E2 -7161.541} C_VEL
LIN {X 0,Y 474.623,Z 286.359,A -85,B 0,C 180,E1 -7164.725,E2 -7164.725} C_VEL
LIN {X 0,Y 474.633,Z 286.363,A -85,B 0,C 180,E1 -7167.787,E2 -7167.787} C_VEL
LIN {X 0,Y 474.611,Z 286.36,A -85,B 0,C 180,E1 -7170.889,E2 -7170.889} C_VEL
LIN {X 0,Y 474.586,Z 286.371,A -85,B 0,C 180,E1 -7173.624,E2 -7173.624} C_VEL
LIN {X 0,Y 474.639,Z 286.357,A -85,B 0,C 180,E1 -7176.642,E2 -7176.642} C_VEL
LIN {X 0,Y 474.656,Z 286.36,A -85,B 0,C 180,E1 -7180.089,E2 -7180.089} C_VEL
LIN {X 0,Y 474.632,Z 286.358,A -85,B 0,C 180,E1 -7182.773,E2 -7182.773} C_VEL
LIN {X 0,Y 474.645,Z 286.358,A -85,B 0,C 180,E1 -7185.421,E2 -7185.421} C_VEL
LIN {X 0,Y 474.698,Z 286.358,A -85,B 0,C 180,E1 -7188.037,E2 -7188.037} C_VEL
LIN {X 0,Y 474.672,Z 286.354,A -85,B 0,C 180,E1 -7191.485,E2 -7191.485} C_VEL
LIN {X 0,Y 474.742,Z 286.351,A -85,B 0,C 180,E1 -7194.052,E2 -7194.052} C_VEL
LIN {X 0,Y 474.876,Z 286.327,A -85,B 0,C 180,E1 -7197.455,E2 -7197.455} C_VEL
LIN {X 0,Y 474.883,Z 286.331,A -85,B 0,C 180,E1 -7200,E2 -7200} C_VEL
LIN {X 0,Y 474.875,Z 286.333,A -85,B 0,C 180,E1 -7202.545,E2 -7202.545} C_VEL
LIN {X 0,Y 474.74,Z 286.346,A -85,B 0,C 180,E1 -7205.948,E2 -7205.948} C_VEL
LIN {X 0,Y 474.664,Z 286.362,A -85,B 0,C 180,E1 -7208.514,E2 -7208.514} C_VEL
LIN {X 0,Y 474.696,Z 286.351,A -85,B 0,C 180,E1 -7211.962,E2 -7211.962} C_VEL
LIN {X 0,Y 474.701,Z 286.349,A -85,B 0,C 180,E1 -7215.455,E2 -7215.455} C_VEL
LIN {X 0,Y 474.661,Z 286.358,A -85,B 0,C 180,E1 -7219.01,E2 -7219.01} C_VEL
LIN {X 0,Y 474.591,Z 286.362,A -85,B 0,C 180,E1 -7221.729,E2 -7221.729} C_VEL
LIN {X 0,Y 474.628,Z 286.362,A -85,B 0,C 180,E1 -7224.495,E2 -7224.495} C_VEL
LIN {X 0,Y 474.6,Z 286.364,A -85,B 0,C 180,E1 -7227.326,E2 -7227.326} C_VEL
LIN {X 0,Y 474.588,Z 286.364,A -85,B 0,C 180,E1 -7230.231,E2 -7230.231} C_VEL
LIN {X 0,Y 474.617,Z 286.365,A -85,B 0,C 180,E1 -7233.222,E2 -7233.222} C_VEL
LIN {X 0,Y 474.587,Z 286.364,A -85,B 0,C 180,E1 -7236.324,E2 -7236.324} C_VEL
LIN {X 0,Y 474.624,Z 286.362,A -85,B 0,C 180,E1 -7239.548,E2 -7239.548} C_VEL
LIN {X 0,Y 474.579,Z 286.364,A -85,B 0,C 180,E1 -7242.23,E2 -7242.23} C_VEL
LIN {X 0,Y 474.619,Z 286.368,A -85,B 0,C 180,E1 -7245.298,E2 -7245.298} C_VEL
LIN {X 0,Y 474.594,Z 286.362,A -85,B 0,C 180,E1 -7248.211,E2 -7248.211} C_VEL
LIN {X 0,Y 474.602,Z 286.368,A -85,B 0,C 180,E1 -7251.541,E2 -7251.541} C_VEL
LIN {X 0,Y 474.621,Z 286.359,A -85,B 0,C 180,E1 -7254.725,E2 -7254.725} C_VEL
LIN {X 0,Y 474.63,Z 286.365,A -85,B 0,C 180,E1 -7257.787,E2 -7257.787} C_VEL
LIN {X 0,Y 474.609,Z 286.363,A -85,B 0,C 180,E1 -7260.888,E2 -7260.888} C_VEL
LIN {X 0,Y 474.644,Z 286.516,A -85,B 0,C 180,E1 -7263.849,E2 -7263.849} C_VEL
LIN {X 0,Y 476.825,Z 297.985,A -85,B 0,C 180,E1 -7265.892,E2 -7265.892} C_VEL
LIN {X 0,Y 476.249,Z 313.702,A -85,B 0,C 180,E1 -7268.498,E2 -7268.498} C_VEL
LIN {X 0,Y 475.567,Z 333.22,A -85,B 0,C 180,E1 -7271.697,E2 -7271.697} C_VEL
LIN {X 0,Y 475.232,Z 342.9,A -85,B 0,C 180,E1 -7273.27,E2 -7273.27} C_VEL
LIN {X 0,Y 477.939,Z 361.914,A -85,B 0,C 180,E1 -7273.655,E2 -7273.655} C_VEL
LIN {X 0,Y 477.293,Z 451.187,A -85,B 0,C 180,E1 -7275.012,E2 -7275.012} C_VEL
LIN {X 0,Y 476.954,Z 463.867,A -85,B 0,C 180,E1 -7275.356,E2 -7275.356} C_VEL
LIN {X 0,Y 476.506,Z 477.463,A -85,B 0,C 180,E1 -7275.915,E2 -7275.915} C_VEL
LIN {X 0,Y 476.073,Z 489.181,A -85,B 0,C 180,E1 -7276.576,E2 -7276.576} C_VEL
LIN {X 0,Y 475.666,Z 499.951,A -85,B 0,C 180,E1 -7277.358,E2 -7277.358} C_VEL
LIN {X 0,Y 475.185,Z 511.154,A -85,B 0,C 180,E1 -7278.374,E2 -7278.374} C_VEL
LIN {X 0,Y 474.737,Z 519.774,A -85,B 0,C 180,E1 -7279.335,E2 -7279.335} C_VEL
LIN {X 0,Y 474.428,Z 527.727,A -85,B 0,C 180,E1 -7280.406,E2 -7280.406} C_VEL
LIN {X 0,Y 474.138,Z 535.496,A -85,B 0,C 180,E1 -7281.69,E2 -7281.69} C_VEL
LIN {X 0,Y 473.901,Z 542.643,A -85,B 0,C 180,E1 -7283.186,E2 -7283.186} C_VEL
LIN {X 0,Y 473.844,Z 547.405,A -85,B 0,C 180,E1 -7284.467,E2 -7284.467} C_VEL
LIN {X 0,Y 473.737,Z 551.038,A -85,B 0,C 180,E1 -7285.746,E2 -7285.746} C_VEL
LIN {X 0,Y 473.796,Z 552.917,A -85,B 0,C 180,E1 -7286.598,E2 -7286.598} C_VEL
LIN {X 0,Y 473.761,Z 554.322,A -85,B 0,C 180,E1 -7287.449,E2 -7287.449} C_VEL
LIN {X 0,Y 473.756,Z 555.324,A -85,B 0,C 180,E1 -7288.299,E2 -7288.299} C_VEL
LIN {X 0,Y 473.675,Z 556.151,A -85,B 0,C 180,E1 -7289.999,E2 -7289.999} C_VEL
LIN {X 0,Y 473.755,Z 555.327,A -85,B 0,C 180,E1 -7291.7,E2 -7291.7} C_VEL
LIN {X 0,Y 473.801,Z 552.927,A -85,B 0,C 180,E1 -7293.401,E2 -7293.401} C_VEL
LIN {X 0,Y 473.762,Z 549.977,A -85,B 0,C 180,E1 -7294.679,E2 -7294.679} C_VEL
LIN {X 0,Y 473.83,Z 545.991,A -85,B 0,C 180,E1 -7295.959,E2 -7295.959} C_VEL
LIN {X 0,Y 474.013,Z 539.873,A -85,B 0,C 180,E1 -7297.454,E2 -7297.454} C_VEL
LIN {X 0,Y 474.219,Z 533.187,A -85,B 0,C 180,E1 -7298.737,E2 -7298.737} C_VEL
LIN {X 0,Y 474.528,Z 524.903,A -85,B 0,C 180,E1 -7300.021,E2 -7300.021} C_VEL
LIN {X 0,Y 474.973,Z 516.438,A -85,B 0,C 180,E1 -7301.09,E2 -7301.09} C_VEL
LIN {X 0,Y 475.419,Z 506.25,A -85,B 0,C 180,E1 -7302.136,E2 -7302.136} C_VEL
LIN {X 0,Y 475.915,Z 494.389,A -85,B 0,C 180,E1 -7303.112,E2 -7303.112} C_VEL
LIN {X 0,Y 476.395,Z 482.522,A -85,B 0,C 180,E1 -7303.87,E2 -7303.87} C_VEL
LIN {X 0,Y 476.862,Z 470.364,A -85,B 0,C 180,E1 -7304.455,E2 -7304.455} C_VEL
LIN {X 0,Y 477.269,Z 457.115,A -85,B 0,C 180,E1 -7304.906,E2 -7304.906} C_VEL
LIN {X 0,Y 477.547,Z 444.095,A -85,B 0,C 180,E1 -7305.169,E2 -7305.169} C_VEL
LIN {X 0,Y 478.05,Z 361.015,A -85,B 0,C 180,E1 -7306.432,E2 -7306.432} C_VEL
LIN {X 0,Y 475.267,Z 342.623,A -85,B 0,C 180,E1 -7306.842,E2 -7306.842} C_VEL
LIN {X 0,Y 476.015,Z 322.959,A -85,B 0,C 180,E1 -7310.076,E2 -7310.076} C_VEL
LIN {X 0,Y 476.689,Z 305.464,A -85,B 0,C 180,E1 -7312.997,E2 -7312.997} C_VEL
LIN {X 0,Y 476.991,Z 298.837,A -85,B 0,C 180,E1 -7314.115,E2 -7314.115} C_VEL
LIN {X 0,Y 475.194,Z 288.962,A -85,B 0,C 180,E1 -7315.92,E2 -7315.92} C_VEL
LIN {X 0,Y 474.627,Z 286.367,A -85,B 0,C 180,E1 -7316.432,E2 -7316.432} C_VEL
LIN {X 0,Y 474.605,Z 286.37,A -85,B 0,C 180,E1 -7319.252,E2 -7319.252} C_VEL
LIN {X 0,Y 474.612,Z 286.369,A -85,B 0,C 180,E1 -7322.43,E2 -7322.43} C_VEL
LIN {X 0,Y 474.608,Z 286.365,A -85,B 0,C 180,E1 -7325.468,E2 -7325.468} C_VEL
LIN {X 0,Y 474.607,Z 286.369,A -85,B 0,C 180,E1 -7328.457,E2 -7328.457} C_VEL
LIN {X 0,Y 474.618,Z 286.36,A -85,B 0,C 180,E1 -7331.785,E2 -7331.785} C_VEL
LIN {X 0,Y 474.614,Z 286.366,A -85,B 0,C 180,E1 -7334.702,E2 -7334.702} C_VEL
LIN {X 0,Y 474.622,Z 286.361,A -85,B 0,C 180,E1 -7337.763,E2 -7337.763} C_VEL
LIN {X 0,Y 474.642,Z 286.364,A -85,B 0,C 180,E1 -7340.454,E2 -7340.454} C_VEL
LIN {X 0,Y 474.585,Z 286.364,A -85,B 0,C 180,E1 -7343.676,E2 -7343.676} C_VEL
LIN {X 0,Y 474.622,Z 286.364,A -85,B 0,C 180,E1 -7346.778,E2 -7346.778} C_VEL
LIN {X 0,Y 474.601,Z 286.361,A -85,B 0,C 180,E1 -7349.77,E2 -7349.77} C_VEL
LIN {X 0,Y 474.694,Z 286.355,A -85,B 0,C 180,E1 -7352.68,E2 -7352.68} C_VEL
LIN {X 0,Y 474.637,Z 286.354,A -85,B 0,C 180,E1 -7355.506,E2 -7355.506} C_VEL
LIN {X 0,Y 474.667,Z 286.352,A -85,B 0,C 180,E1 -7359.185,E2 -7359.185} C_VEL
LIN {X 0,Y 474.654,Z 286.356,A -85,B 0,C 180,E1 -7361.884,E2 -7361.884} C_VEL
LIN {X 0,Y 474.697,Z 286.352,A -85,B 0,C 180,E1 -7364.544,E2 -7364.544} C_VEL
LIN {X 0,Y 474.701,Z 286.347,A -85,B 0,C 180,E1 -7368.038,E2 -7368.038} C_VEL
LIN {X 0,Y 474.725,Z 286.345,A -85,B 0,C 180,E1 -7371.487,E2 -7371.487} C_VEL
LIN {X 0,Y 474.775,Z 286.341,A -85,B 0,C 180,E1 -7374.053,E2 -7374.053} C_VEL
LIN {X 0,Y 474.892,Z 286.327,A -85,B 0,C 180,E1 -7377.456,E2 -7377.456} C_VEL
LIN {X 0,Y 474.909,Z 286.322,A -85,B 0,C 180,E1 -7380,E2 -7380} C_VEL
LIN {X 0,Y 474.891,Z 286.328,A -85,B 0,C 180,E1 -7382.545,E2 -7382.545} C_VEL
LIN {X 0,Y 474.775,Z 286.339,A -85,B 0,C 180,E1 -7385.948,E2 -7385.948} C_VEL
LIN {X 0,Y 474.725,Z 286.348,A -85,B 0,C 180,E1 -7388.514,E2 -7388.514} C_VEL
LIN {X 0,Y 474.701,Z 286.349,A -85,B 0,C 180,E1 -7391.963,E2 -7391.963} C_VEL
LIN {X 0,Y 474.697,Z 286.353,A -85,B 0,C 180,E1 -7395.456,E2 -7395.456} C_VEL
LIN {X 0,Y 474.66,Z 286.36,A -85,B 0,C 180,E1 -7399.011,E2 -7399.011} C_VEL
LIN {X 0,Y 474.586,Z 286.364,A -85,B 0,C 180,E1 -7401.729,E2 -7401.729} C_VEL
LIN {X 0,Y 474.636,Z 286.358,A -85,B 0,C 180,E1 -7404.495,E2 -7404.495} C_VEL
LIN {X 0,Y 474.678,Z 286.359,A -85,B 0,C 180,E1 -7407.335,E2 -7407.335} C_VEL
LIN {X 0,Y 474.601,Z 286.365,A -85,B 0,C 180,E1 -7410.81,E2 -7410.81} C_VEL
LIN {X 0,Y 474.623,Z 286.364,A -85,B 0,C 180,E1 -7413.222,E2 -7413.222} C_VEL
LIN {X 0,Y 474.587,Z 286.363,A -85,B 0,C 180,E1 -7416.324,E2 -7416.324} C_VEL
LIN {X 0,Y 474.622,Z 286.365,A -85,B 0,C 180,E1 -7419.549,E2 -7419.549} C_VEL
LIN {X 0,Y 474.589,Z 286.364,A -85,B 0,C 180,E1 -7422.233,E2 -7422.233} C_VEL
LIN {X 0,Y 474.615,Z 286.368,A -85,B 0,C 180,E1 -7425.299,E2 -7425.299} C_VEL
LIN {X 0,Y 474.6,Z 286.364,A -85,B 0,C 180,E1 -7428.213,E2 -7428.213} C_VEL
LIN {X 0,Y 474.6,Z 286.37,A -85,B 0,C 180,E1 -7431.542,E2 -7431.542} C_VEL
LIN {X 0,Y 474.62,Z 286.359,A -85,B 0,C 180,E1 -7434.726,E2 -7434.726} C_VEL
LIN {X 0,Y 474.634,Z 286.365,A -85,B 0,C 180,E1 -7437.788,E2 -7437.788} C_VEL
LIN {X 0,Y 474.666,Z 286.473,A -85,B 0,C 180,E1 -7441.267,E2 -7441.267} C_VEL
LIN {X 0,Y 475.556,Z 292.325,A -85,B 0,C 180,E1 -7442.464,E2 -7442.464} C_VEL
LIN {X 0,Y 475.48,Z 301.578,A -85,B 0,C 180,E1 -7444.237,E2 -7444.237} C_VEL
LIN {X 0,Y 478.309,Z 315.335,A -85,B 0,C 180,E1 -7444.564,E2 -7444.564} C_VEL
LIN {X 0,Y 477.964,Z 357.805,A -85,B 0,C 180,E1 -7445.209,E2 -7445.209} C_VEL
